C05452=1120.411,381.340,-87.972,-176.855,11.261,149.470
C05453=1120.415,381.092,-87.935,-176.859,11.258,149.470
C05454=1120.418,380.845,-87.897,-176.861,11.255,149.470
C05455=1120.423,380.598,-87.860,-176.865,11.253,149.470
C05456=1120.426,380.351,-87.822,-176.868,11.250,149.470
C05457=1120.430,380.103,-87.786,-176.871,11.248,149.471
C05458=1120.434,379.857,-87.748,-176.873,11.246,149.471
C05459=1120.437,379.609,-87.711,-176.876,11.243,149.471
C05460=1120.441,379.362,-87.673,-176.880,11.241,149.471
C05461=1120.444,379.115,-87.636,-176.883,11.238,149.471
C05462=1120.449,378.867,-87.599,-176.886,11.235,149.471
C05463=1120.452,378.621,-87.562,-176.889,11.233,149.471
C05464=1120.456,378.373,-87.524,-176.892,11.230,149.471
C05465=1120.460,378.126,-87.487,-176.895,11.228,149.472
C05466=1120.464,377.879,-87.450,-176.898,11.226,149.472
C05467=1120.467,377.631,-87.413,-176.901,11.223,149.472
C05468=1120.471,377.385,-87.375,-176.904,11.221,149.472
C05469=1120.475,377.138,-87.338,-176.908,11.218,149.472
C05470=1120.479,376.890,-87.301,-176.910,11.215,149.472
C05471=1120.482,376.643,-87.264,-176.913,11.214,149.473
C05472=1120.485,376.430,-87.232,-176.916,11.211,149.473
C05473=1120.489,376.219,-87.201,-176.919,11.209,149.473
C05474=1120.491,376.007,-87.169,-176.921,11.207,149.473
C05475=1120.495,375.795,-87.136,-176.924,11.205,149.473
C05476=1120.498,375.582,-87.105,-176.927,11.203,149.473
C05477=1120.501,375.371,-87.073,-176.929,11.201,149.473
C05478=1120.504,375.159,-87.041,-176.933,11.198,149.474
C05479=1120.508,374.946,-87.009,-176.935,11.197,149.474
C05480=1120.511,374.699,-86.973,-176.938,11.194,149.474
C05481=1120.515,374.452,-86.935,-176.941,11.191,149.474
C05482=1120.519,374.205,-86.899,-176.944,11.190,149.474
C05483=1120.523,373.957,-86.861,-176.947,11.187,149.474
C05484=1120.527,373.710,-86.824,-176.951,11.185,149.475
C05485=1120.530,373.463,-86.788,-176.954,11.182,149.475
C05486=1120.534,373.215,-86.751,-176.957,11.180,149.475
C05487=1120.538,372.968,-86.714,-176.961,11.177,149.475
C05488=1120.542,372.721,-86.677,-176.964,11.175,149.475
C05489=1120.546,372.474,-86.640,-176.967,11.173,149.476
C05490=1120.549,372.227,-86.603,-176.970,11.171,149.476
C05491=1120.552,371.980,-86.566,-176.973,11.168,149.476
C05492=1120.556,371.732,-86.529,-176.976,11.166,149.476
C05493=1120.561,371.485,-86.492,-176.980,11.163,149.477
C05494=1120.564,371.238,-86.456,-176.983,11.161,149.477
C05495=1120.567,370.990,-86.419,-176.986,11.158,149.477
C05496=1120.571,370.743,-86.382,-176.989,11.157,149.477
C05497=1120.575,370.496,-86.347,-176.992,11.154,149.477
C05498=1120.579,370.249,-86.310,-176.996,11.152,149.478
C05499=1120.583,370.001,-86.273,-176.999,11.149,149.478
C05500=1120.586,369.754,-86.236,-177.002,11.147,149.478
C05501=1120.590,369.507,-86.199,-177.005,11.144,149.478
C05502=1120.594,369.259,-86.163,-177.009,11.142,149.478
C05503=1120.598,369.012,-86.126,-177.012,11.139,149.479
C05504=1120.602,368.765,-86.089,-177.015,11.137,149.479
C05505=1120.606,368.518,-86.053,-177.018,11.135,149.479
C05506=1120.609,368.271,-86.017,-177.021,11.133,149.479
C05507=1120.613,368.023,-85.980,-177.025,11.130,149.480
C05508=1120.616,367.776,-85.944,-177.028,11.128,149.480
C05509=1120.620,367.529,-85.907,-177.032,11.125,149.480
C05510=1120.625,367.281,-85.870,-177.035,11.123,149.480
C05511=1120.628,367.034,-85.834,-177.038,11.121,149.481
C05512=1120.632,366.787,-85.797,-177.042,11.118,149.481
C05513=1120.636,366.540,-85.761,-177.045,11.116,149.481
C05514=1120.640,366.292,-85.725,-177.048,11.113,149.481
C05515=1120.643,366.044,-85.688,-177.052,11.111,149.482
C05516=1120.647,365.797,-85.651,-177.055,11.109,149.482
C05517=1120.651,365.550,-85.616,-177.058,11.107,149.482
C05518=1120.655,365.303,-85.579,-177.061,11.104,149.482
C05519=1120.658,365.056,-85.543,-177.064,11.102,149.482
C05520=1120.662,364.808,-85.507,-177.068,11.099,149.483
C05521=1120.666,364.561,-85.470,-177.071,11.097,149.483
C05522=1120.670,364.314,-85.434,-177.075,11.095,149.483
C05523=1120.674,364.066,-85.398,-177.078,11.092,149.483
C05524=1120.678,363.819,-85.361,-177.081,11.090,149.484
C05525=1120.681,363.572,-85.326,-177.085,11.087,149.484
C05526=1120.685,363.324,-85.289,-177.088,11.085,149.484
C05527=1120.689,363.077,-85.253,-177.092,11.083,149.485
C05528=1120.692,362.864,-85.222,-177.094,11.081,149.485
C05529=1120.696,362.652,-85.191,-177.098,11.079,149.485
C05530=1120.699,362.440,-85.160,-177.100,11.077,149.485
C05531=1120.702,362.228,-85.129,-177.103,11.075,149.485
C05532=1120.705,362.015,-85.098,-177.106,11.072,149.486
C05533=1120.708,361.803,-85.067,-177.109,11.071,149.486
C05534=1120.711,361.591,-85.036,-177.112,11.068,149.486
C05535=1120.715,361.379,-85.005,-177.115,11.067,149.486
C05536=1120.718,361.132,-84.969,-177.118,11.064,149.486
C05537=1120.723,360.884,-84.933,-177.121,11.062,149.487
C05538=1120.726,360.637,-84.897,-177.125,11.059,149.487
C05539=1120.730,360.390,-84.861,-177.128,11.057,149.487
C05540=1120.734,360.142,-84.825,-177.131,11.055,149.488
C05541=1120.738,359.895,-84.789,-177.135,11.052,149.488
C05542=1120.741,359.648,-84.753,-177.138,11.050,149.488
C05543=1120.745,359.400,-84.717,-177.142,11.047,149.488
C05544=1120.749,359.152,-84.681,-177.145,11.045,149.489
C05545=1120.753,358.905,-84.646,-177.148,11.043,149.489
C05546=1120.756,358.658,-84.609,-177.152,11.040,149.489
C05547=1120.761,358.410,-84.573,-177.155,11.038,149.489
C05548=1120.764,358.163,-84.538,-177.159,11.035,149.490
C05549=1120.768,357.915,-84.502,-177.162,11.033,149.490
C05550=1120.771,357.668,-84.466,-177.165,11.031,149.490
C05551=1120.775,357.421,-84.430,-177.169,11.028,149.490
C05552=1120.780,357.174,-84.395,-177.173,11.025,149.491
C05553=1120.784,356.926,-84.359,-177.176,11.023,149.491
C05554=1120.787,356.679,-84.323,-177.180,11.020,149.491
C05555=1120.791,356.431,-84.288,-177.183,11.018,149.491
C05556=1120.795,356.184,-84.252,-177.187,11.016,149.492
C05557=1120.799,355.936,-84.216,-177.190,11.013,149.492
C05558=1120.803,355.688,-84.181,-177.193,11.011,149.492
C05559=1120.806,355.441,-84.144,-177.197,11.008,149.492
C05560=1120.810,355.195,-84.109,-177.200,11.006,149.493
C05561=1120.814,354.947,-84.074,-177.204,11.004,149.493
C05562=1120.818,354.700,-84.038,-177.207,11.001,149.493
C05563=1120.821,354.452,-84.003,-177.211,10.998,149.493
C05564=1120.825,354.205,-83.967,-177.214,10.995,149.494
C05565=1120.829,353.957,-83.931,-177.217,10.993,149.494
C05566=1120.834,353.709,-83.896,-177.221,10.991,149.494
C05567=1120.838,353.462,-83.861,-177.224,10.988,149.495
C05568=1120.841,353.214,-83.825,-177.228,10.986,149.495
C05569=1120.845,352.967,-83.790,-177.231,10.983,149.495
C05570=1120.849,352.719,-83.754,-177.235,10.980,149.495
C05571=1120.852,352.472,-83.719,-177.239,10.978,149.496
C05572=1120.857,352.225,-83.683,-177.242,10.976,149.496
C05573=1120.860,351.978,-83.648,-177.245,10.973,149.496
C05574=1120.864,351.729,-83.613,-177.249,10.971,149.496
C05575=1120.868,351.482,-83.578,-177.252,10.968,149.496
C05576=1120.872,351.235,-83.542,-177.256,10.965,149.497
C05577=1120.876,350.988,-83.507,-177.259,10.963,149.497
C05578=1120.879,350.740,-83.471,-177.263,10.960,149.497
C05579=1120.883,350.492,-83.436,-177.266,10.958,149.498
C05580=1120.888,350.245,-83.401,-177.270,10.955,149.498
C05581=1120.891,349.998,-83.366,-177.273,10.952,149.498
C05582=1120.895,349.750,-83.331,-177.277,10.950,149.498
C05583=1120.899,349.502,-83.295,-177.280,10.947,149.498
C05584=1120.902,349.290,-83.266,-177.283,10.945,149.499
C05585=1120.906,349.078,-83.235,-177.286,10.943,149.499
C05586=1120.909,348.866,-83.205,-177.288,10.941,149.499
C05587=1120.912,348.652,-83.175,-177.291,10.938,149.499
C05588=1120.916,348.440,-83.145,-177.294,10.937,149.499
C05589=1120.919,348.228,-83.114,-177.297,10.935,149.500
C05590=1120.923,348.016,-83.085,-177.300,10.932,149.500
C05591=1120.926,347.803,-83.054,-177.302,10.931,149.500
C05592=1120.929,347.556,-83.019,-177.306,10.928,149.500
C05593=1120.933,347.308,-82.985,-177.309,10.926,149.500
C05594=1120.938,347.061,-82.949,-177.312,10.923,149.500
C05595=1120.942,346.813,-82.915,-177.315,10.920,149.501
C05596=1120.945,346.566,-82.879,-177.318,10.918,149.501
C05597=1120.950,346.318,-82.845,-177.322,10.915,149.501
C05598=1120.953,346.071,-82.810,-177.325,10.913,149.501
C05599=1120.957,345.823,-82.775,-177.328,10.911,149.501
C05600=1120.961,345.576,-82.740,-177.331,10.908,149.502
C05601=1120.965,345.328,-82.705,-177.335,10.905,149.502
C05602=1120.969,345.080,-82.670,-177.337,10.904,149.502
C05603=1120.972,344.833,-82.635,-177.341,10.901,149.502
C05604=1120.976,344.585,-82.601,-177.344,10.899,149.502
C05605=1120.981,344.338,-82.565,-177.347,10.896,149.503
C05606=1120.985,344.090,-82.531,-177.350,10.893,149.503
C05607=1120.988,343.843,-82.497,-177.353,10.891,149.503
C05608=1120.992,343.596,-82.461,-177.357,10.889,149.503
C05609=1120.996,343.348,-82.426,-177.360,10.886,149.503
C05610=1121.001,343.100,-82.392,-177.363,10.884,149.504
C05611=1121.004,342.852,-82.358,-177.367,10.881,149.504
C05612=1121.008,342.606,-82.322,-177.370,10.878,149.504
C05613=1121.012,342.357,-82.288,-177.373,10.876,149.504
C05614=1121.016,342.110,-82.254,-177.376,10.873,149.504
C05615=1121.020,341.862,-82.219,-177.380,10.871,149.505
C05616=1121.024,341.615,-82.183,-177.383,10.869,149.505
C05617=1121.027,341.368,-82.149,-177.385,10.867,149.505
C05618=1121.031,341.120,-82.115,-177.388,10.864,149.505
C05619=1121.036,340.872,-82.080,-177.392,10.862,149.505
C05620=1121.039,340.624,-82.046,-177.395,10.859,149.506
C05621=1121.043,340.377,-82.011,-177.398,10.857,149.506
C05622=1121.047,340.129,-81.976,-177.401,10.854,149.506
C05623=1121.051,339.882,-81.942,-177.405,10.851,149.506
C05624=1121.055,339.634,-81.907,-177.408,10.849,149.506
C05625=1121.059,339.387,-81.873,-177.411,10.847,149.507
C05626=1121.063,339.139,-81.838,-177.414,10.844,149.507
C05627=1121.068,338.891,-81.804,-177.417,10.841,149.507
C05628=1121.071,338.644,-81.770,-177.421,10.839,149.507
C05629=1121.075,338.396,-81.735,-177.424,10.836,149.507
C05630=1121.079,338.149,-81.701,-177.427,10.834,149.508
C05631=1121.083,337.901,-81.667,-177.430,10.831,149.508
C05632=1121.087,337.654,-81.633,-177.433,10.830,149.508
C05633=1121.091,337.406,-81.598,-177.436,10.827,149.508
C05634=1121.095,337.159,-81.564,-177.440,10.825,149.508
C05635=1121.099,336.911,-81.529,-177.443,10.822,149.508
C05636=1121.103,336.663,-81.495,-177.446,10.819,149.509
C05637=1121.107,336.415,-81.460,-177.449,10.817,149.509
C05638=1121.110,336.168,-81.427,-177.453,10.814,149.509
C05639=1121.115,335.921,-81.392,-177.455,10.812,149.509
C05640=1121.119,335.708,-81.363,-177.458,10.810,149.510
C05641=1121.122,335.496,-81.334,-177.461,10.807,149.510
C05642=1121.125,335.283,-81.305,-177.464,10.806,149.510
C05643=1121.128,335.070,-81.275,-177.467,10.803,149.510
C05644=1121.131,334.858,-81.245,-177.469,10.801,149.510
C05645=1121.135,334.645,-81.216,-177.472,10.799,149.510
C05646=1121.138,334.432,-81.187,-177.475,10.797,149.510
C05647=1121.141,334.220,-81.158,-177.477,10.795,149.511
C05648=1121.145,333.972,-81.124,-177.481,10.792,149.511
C05649=1121.150,333.725,-81.089,-177.484,10.790,149.511
C05650=1121.153,333.477,-81.056,-177.487,10.787,149.511
C05651=1121.158,333.229,-81.022,-177.490,10.784,149.511
C05652=1121.162,332.982,-80.988,-177.493,10.782,149.512
C05653=1121.165,332.734,-80.953,-177.497,10.780,149.512
C05654=1121.170,332.486,-80.920,-177.500,10.777,149.512
C05655=1121.174,332.239,-80.886,-177.502,10.775,149.512
C05656=1121.177,331.991,-80.852,-177.506,10.773,149.512
C05657=1121.181,331.744,-80.818,-177.509,10.770,149.513
C05658=1121.186,331.496,-80.784,-177.512,10.767,149.513
C05659=1121.189,331.248,-80.750,-177.515,10.765,149.513
C05660=1121.193,331.001,-80.717,-177.519,10.763,149.513
C05661=1121.198,330.753,-80.682,-177.522,10.760,149.513
C05662=1121.201,330.505,-80.649,-177.525,10.757,149.513
C05663=1121.205,330.258,-80.615,-177.528,10.755,149.514
C05664=1121.209,330.010,-80.582,-177.531,10.752,149.514
C05665=1121.213,329.762,-80.547,-177.534,10.750,149.514
C05666=1121.217,329.514,-80.514,-177.538,10.747,149.514
C05667=1121.221,329.267,-80.480,-177.541,10.745,149.515
C05668=1121.225,329.019,-80.446,-177.544,10.742,149.515
C05669=1121.228,328.771,-80.412,-177.547,10.740,149.515
C05670=1121.233,328.523,-80.379,-177.550,10.738,149.515
C05671=1121.237,328.276,-80.345,-177.553,10.735,149.515
C05672=1121.241,328.029,-80.311,-177.556,10.733,149.515
C05673=1121.244,327.781,-80.277,-177.560,10.730,149.516
C05674=1121.249,327.533,-80.244,-177.563,10.728,149.516
C05675=1121.253,327.285,-80.211,-177.566,10.725,149.516
C05676=1121.257,327.038,-80.176,-177.569,10.723,149.516
C05677=1121.261,326.789,-80.143,-177.572,10.720,149.516
C05678=1121.265,326.542,-80.110,-177.575,10.717,149.516
C05679=1121.269,326.295,-80.076,-177.579,10.715,149.517
C05680=1121.273,326.047,-80.043,-177.582,10.712,149.517
C05681=1121.277,325.799,-80.010,-177.585,10.710,149.517
C05682=1121.280,325.551,-79.975,-177.588,10.707,149.517
C05683=1121.284,325.304,-79.942,-177.592,10.705,149.518
C05684=1121.289,325.056,-79.909,-177.594,10.703,149.518
C05685=1121.293,324.808,-79.876,-177.597,10.700,149.518
C05686=1121.297,324.561,-79.842,-177.601,10.698,149.518
C05687=1121.300,324.313,-79.809,-177.604,10.695,149.518
C05688=1121.305,324.065,-79.775,-177.607,10.693,149.518
C05689=1121.309,323.817,-79.742,-177.610,10.690,149.519
C05690=1121.313,323.569,-79.708,-177.613,10.688,149.519
C05691=1121.317,323.322,-79.675,-177.616,10.685,149.519
C05692=1121.321,323.074,-79.641,-177.620,10.682,149.519
C05693=1121.324,322.826,-79.608,-177.623,10.680,149.519
C05694=1121.328,322.578,-79.575,-177.626,10.677,149.520
C05695=1121.332,322.331,-79.542,-177.629,10.675,149.520
C05696=1121.336,322.118,-79.513,-177.632,10.673,149.520
C05697=1121.340,321.906,-79.485,-177.634,10.671,149.520
C05698=1121.343,321.693,-79.456,-177.637,10.668,149.520
C05699=1121.346,321.480,-79.428,-177.639,10.666,149.520
C05700=1121.350,321.267,-79.399,-177.643,10.664,149.521
C05701=1121.353,321.054,-79.371,-177.645,10.662,149.521
C05702=1121.357,320.842,-79.343,-177.648,10.660,149.521
C05703=1121.360,320.629,-79.314,-177.651,10.658,149.521
C05704=1121.364,320.382,-79.281,-177.654,10.655,149.521
C05705=1121.368,320.134,-79.248,-177.656,10.653,149.521
C05706=1121.372,319.886,-79.215,-177.660,10.651,149.522
C05707=1121.376,319.638,-79.181,-177.663,10.648,149.522
C05708=1121.380,319.390,-79.148,-177.666,10.645,149.522
C05709=1121.384,319.142,-79.115,-177.669,10.643,149.522
C05710=1121.387,318.895,-79.082,-177.672,10.640,149.522
C05711=1121.391,318.647,-79.049,-177.675,10.638,149.523
C05712=1121.396,318.399,-79.017,-177.679,10.635,149.523
C05713=1121.400,318.151,-78.984,-177.682,10.633,149.523
C05714=1121.404,317.903,-78.951,-177.685,10.630,149.523
C05715=1121.408,317.656,-78.917,-177.688,10.628,149.523
C05716=1121.412,317.408,-78.885,-177.691,10.625,149.523
C05717=1121.416,317.160,-78.852,-177.695,10.622,149.524
C05718=1121.420,316.912,-78.819,-177.698,10.620,149.524
C05719=1121.424,316.664,-78.786,-177.700,10.618,149.524
C05720=1121.428,316.417,-78.754,-177.704,10.616,149.524
C05721=1121.432,316.169,-78.720,-177.706,10.613,149.524
C05722=1121.436,315.922,-78.687,-177.710,10.610,149.525
C05723=1121.441,315.673,-78.655,-177.713,10.608,149.525
C05724=1121.444,315.426,-78.622,-177.716,10.605,149.525
C05725=1121.448,315.178,-78.589,-177.719,10.603,149.525
C05726=1121.453,314.930,-78.557,-177.722,10.600,149.525
C05727=1121.456,314.682,-78.524,-177.726,10.597,149.526
C05728=1121.460,314.435,-78.491,-177.729,10.595,149.526
C05729=1121.465,314.186,-78.458,-177.732,10.592,149.526
C05730=1121.468,313.939,-78.426,-177.735,10.590,149.526
C05731=1121.472,313.691,-78.393,-177.738,10.587,149.526
C05732=1121.477,313.443,-78.360,-177.741,10.585,149.526
C05733=1121.480,313.195,-78.328,-177.744,10.583,149.527
C05734=1121.484,312.947,-78.295,-177.747,10.580,149.527
C05735=1121.489,312.700,-78.263,-177.750,10.578,149.527
C05736=1121.493,312.452,-78.231,-177.753,10.575,149.527
C05737=1121.497,312.204,-78.198,-177.757,10.573,149.527
C05738=1121.501,311.956,-78.166,-177.760,10.570,149.527
C05739=1121.505,311.708,-78.133,-177.763,10.567,149.528
C05740=1121.509,311.460,-78.100,-177.766,10.565,149.528
C05741=1121.513,311.213,-78.068,-177.769,10.562,149.528
C05742=1121.517,310.964,-78.035,-177.773,10.560,149.528
C05743=1121.520,310.717,-78.003,-177.775,10.557,149.528
C05744=1121.525,310.468,-77.970,-177.778,10.555,149.529
C05745=1121.529,310.222,-77.938,-177.781,10.552,149.529
C05746=1121.533,309.973,-77.905,-177.784,10.550,149.529
C05747=1121.537,309.725,-77.874,-177.787,10.547,149.529
C05748=1121.541,309.478,-77.840,-177.791,10.545,149.529
C05749=1121.545,309.230,-77.809,-177.794,10.542,149.530
C05750=1121.549,308.981,-77.776,-177.797,10.540,149.530
C05751=1121.553,308.735,-77.744,-177.800,10.537,149.530
C05752=1121.557,308.521,-77.716,-177.803,10.535,149.530
C05753=1121.560,308.308,-77.688,-177.805,10.532,149.530
C05754=1121.564,308.095,-77.661,-177.808,10.531,149.530
C05755=1121.568,307.882,-77.633,-177.810,10.529,149.530
C05756=1121.571,307.670,-77.605,-177.813,10.526,149.531
C05757=1121.574,307.457,-77.577,-177.816,10.524,149.531
C05758=1121.578,307.244,-77.550,-177.818,10.522,149.531
C05759=1121.582,307.031,-77.522,-177.821,10.520,149.531
C05760=1121.585,306.783,-77.490,-177.825,10.517,149.531
C05761=1121.590,306.535,-77.459,-177.828,10.514,149.531
C05762=1121.594,306.288,-77.425,-177.831,10.512,149.532
C05763=1121.598,306.040,-77.394,-177.834,10.510,149.532
C05764=1121.602,305.791,-77.361,-177.837,10.508,149.532
C05765=1121.606,305.543,-77.329,-177.840,10.505,149.532
C05766=1121.610,305.296,-77.298,-177.843,10.502,149.532
C05767=1121.615,305.048,-77.265,-177.846,10.500,149.533
C05768=1121.618,304.800,-77.234,-177.849,10.497,149.533
C05769=1121.622,304.553,-77.201,-177.852,10.495,149.533
C05770=1121.627,304.304,-77.169,-177.855,10.492,149.533
C05771=1121.630,304.056,-77.137,-177.859,10.489,149.533
C05772=1121.634,303.808,-77.105,-177.862,10.487,149.533
C05773=1121.639,303.561,-77.073,-177.865,10.484,149.534
C05774=1121.643,303.313,-77.041,-177.868,10.482,149.534
C05775=1121.647,303.065,-77.010,-177.871,10.480,149.534
C05776=1121.652,302.817,-76.977,-177.873,10.477,149.534
C05777=1121.655,302.569,-76.946,-177.877,10.475,149.534
C05778=1121.659,302.321,-76.914,-177.880,10.472,149.535
C05779=1121.664,302.073,-76.882,-177.883,10.469,149.535
C05780=1121.668,301.825,-76.850,-177.886,10.467,149.535
C05781=1121.672,301.577,-76.819,-177.889,10.464,149.535
C05782=1121.676,301.329,-76.787,-177.893,10.462,149.535
C05783=1121.681,301.081,-76.755,-177.896,10.459,149.535
C05784=1121.684,300.833,-76.723,-177.899,10.457,149.536
C05785=1121.689,300.586,-76.691,-177.902,10.454,149.536
C05786=1121.692,300.337,-76.660,-177.905,10.451,149.536
C05787=1121.696,300.089,-76.628,-177.908,10.449,149.536
C05788=1121.701,299.842,-76.596,-177.911,10.447,149.536
C05789=1121.705,299.593,-76.565,-177.914,10.444,149.536
C05790=1121.709,299.345,-76.533,-177.917,10.442,149.537
C05791=1121.713,299.098,-76.501,-177.920,10.439,149.537
C05792=1121.717,298.850,-76.469,-177.923,10.437,149.537
C05793=1121.721,298.602,-76.439,-177.926,10.434,149.537
C05794=1121.725,298.354,-76.407,-177.930,10.431,149.537
C05795=1121.729,298.106,-76.375,-177.933,10.429,149.537
C05796=1121.734,297.858,-76.343,-177.936,10.426,149.538
C05797=1121.738,297.609,-76.312,-177.939,10.423,149.538
C05798=1121.742,297.362,-76.280,-177.942,10.422,149.538
C05799=1121.746,297.114,-76.248,-177.945,10.419,149.538
C05800=1121.750,296.865,-76.217,-177.948,10.417,149.538
C05801=1121.754,296.618,-76.186,-177.951,10.414,149.539
C05802=1121.758,296.370,-76.154,-177.954,10.411,149.539
C05803=1121.762,296.122,-76.123,-177.957,10.409,149.539
C05804=1121.766,295.874,-76.091,-177.960,10.406,149.539
C05805=1121.771,295.626,-76.061,-177.963,10.403,149.539
C05806=1121.774,295.378,-76.029,-177.967,10.401,149.540
C05807=1121.779,295.130,-75.998,-177.970,10.398,149.540
C05808=1121.783,294.904,-75.969,-177.972,10.396,149.540
C05809=1121.786,294.679,-75.940,-177.975,10.394,149.540
C05810=1121.790,294.454,-75.912,-177.978,10.392,149.540
C05811=1121.794,294.228,-75.883,-177.980,10.389,149.540
C05812=1121.797,294.003,-75.855,-177.983,10.387,149.541
C05813=1121.801,293.778,-75.827,-177.986,10.385,149.541
C05814=1121.805,293.552,-75.798,-177.988,10.383,149.541
C05815=1121.809,293.327,-75.770,-177.992,10.380,149.541
C05816=1121.813,293.079,-75.739,-177.995,10.378,149.541
C05817=1121.817,292.831,-75.708,-177.998,10.375,149.541
C05818=1121.821,292.583,-75.676,-178.001,10.372,149.541
C05819=1121.825,292.335,-75.646,-178.004,10.370,149.542
C05820=1121.829,292.099,-75.616,-178.007,10.368,149.542
C05821=1121.833,291.863,-75.586,-178.010,10.365,149.542
C05822=1121.837,291.628,-75.556,-178.013,10.363,149.542
C05823=1121.841,291.393,-75.527,-178.015,10.361,149.542
C05824=1121.845,291.157,-75.497,-178.018,10.358,149.543
C05825=1121.848,290.921,-75.467,-178.021,10.356,149.543
C05826=1121.853,290.685,-75.438,-178.024,10.353,149.543
C05827=1121.856,290.450,-75.409,-178.027,10.351,149.543
C05828=1121.861,290.202,-75.378,-178.030,10.348,149.543
C05829=1121.865,289.953,-75.347,-178.033,10.346,149.543
C05830=1121.869,289.706,-75.316,-178.036,10.343,149.543
C05831=1121.873,289.457,-75.284,-178.040,10.341,149.544
C05832=1121.877,289.210,-75.254,-178.043,10.338,149.544
C05833=1121.881,288.962,-75.223,-178.045,10.335,149.544
C05834=1121.886,288.713,-75.192,-178.049,10.333,149.544
C05835=1121.890,288.466,-75.161,-178.051,10.331,149.544
C05836=1121.894,288.217,-75.130,-178.054,10.328,149.545
C05837=1121.898,287.969,-75.100,-178.057,10.326,149.545
C05838=1121.902,287.721,-75.069,-178.061,10.323,149.545
C05839=1121.906,287.473,-75.038,-178.064,10.320,149.545
C05840=1121.910,287.225,-75.008,-178.067,10.318,149.545
C05841=1121.914,286.976,-74.976,-178.070,10.315,149.545
C05842=1121.919,286.729,-74.945,-178.073,10.313,149.546
C05843=1121.923,286.481,-74.914,-178.076,10.310,149.546
C05844=1121.926,286.233,-74.884,-178.079,10.307,149.546
C05845=1121.931,285.985,-74.853,-178.082,10.306,149.546
C05846=1121.936,285.737,-74.822,-178.085,10.303,149.546
C05847=1121.939,285.489,-74.792,-178.088,10.301,149.547
C05848=1121.944,285.241,-74.761,-178.091,10.298,149.547
C05849=1121.948,284.993,-74.730,-178.094,10.295,149.547
C05850=1121.951,284.744,-74.699,-178.097,10.293,149.547
C05851=1121.956,284.496,-74.669,-178.100,10.290,149.547
C05852=1121.960,284.249,-74.639,-178.104,10.287,149.547
C05853=1121.965,284.001,-74.608,-178.107,10.285,149.547
C05854=1121.969,283.752,-74.577,-178.109,10.283,149.548
C05855=1121.973,283.504,-74.547,-178.112,10.280,149.548
C05856=1121.977,283.256,-74.516,-178.115,10.277,149.548
C05857=1121.981,283.007,-74.486,-178.119,10.275,149.548
C05858=1121.985,282.759,-74.455,-178.121,10.272,149.548
C05859=1121.990,282.512,-74.424,-178.125,10.270,149.549
C05860=1121.994,282.264,-74.394,-178.128,10.267,149.549
C05861=1121.998,282.015,-74.363,-178.131,10.264,149.549
C05862=1122.002,281.767,-74.334,-178.134,10.262,149.549
C05863=1122.007,281.519,-74.303,-178.136,10.260,149.549
C05864=1122.010,281.306,-74.277,-178.140,10.258,149.550
C05865=1122.014,281.093,-74.250,-178.143,10.255,149.550
C05866=1122.017,280.880,-74.225,-178.145,10.253,149.550
C05867=1122.021,280.666,-74.198,-178.148,10.250,149.550
C05868=1122.024,280.453,-74.173,-178.151,10.248,149.550
C05869=1122.028,280.240,-74.146,-178.154,10.246,149.550
C05870=1122.031,280.027,-74.120,-178.157,10.243,149.551
C05871=1122.036,279.813,-74.094,-178.160,10.240,149.551
C05872=1122.039,279.566,-74.064,-178.163,10.238,149.551
C05873=1122.043,279.318,-74.034,-178.166,10.235,149.551
C05874=1122.048,279.070,-74.004,-178.169,10.233,149.551
C05875=1122.051,278.821,-73.973,-178.172,10.230,149.551
C05876=1122.056,278.573,-73.943,-178.176,10.227,149.552
C05877=1122.060,278.325,-73.913,-178.179,10.224,149.552
C05878=1122.064,278.077,-73.883,-178.183,10.222,149.552
C05879=1122.069,277.829,-73.853,-178.186,10.219,149.552
C05880=1122.072,277.580,-73.822,-178.188,10.216,149.552
C05881=1122.077,277.332,-73.792,-178.192,10.214,149.553
C05882=1122.081,277.084,-73.762,-178.195,10.211,149.553
C05883=1122.085,276.837,-73.732,-178.198,10.208,149.553
C05884=1122.090,276.588,-73.702,-178.201,10.206,149.553
C05885=1122.094,276.340,-73.672,-178.205,10.202,149.553
C05886=1122.098,276.092,-73.642,-178.208,10.200,149.553
C05887=1122.102,275.844,-73.612,-178.211,10.197,149.553
C05888=1122.106,275.595,-73.582,-178.214,10.194,149.554
C05889=1122.110,275.347,-73.552,-178.217,10.192,149.554
C05890=1122.114,275.099,-73.522,-178.220,10.189,149.554
C05891=1122.119,274.851,-73.492,-178.223,10.186,149.554
C05892=1122.123,274.603,-73.462,-178.226,10.184,149.554
C05893=1122.127,274.355,-73.433,-178.229,10.181,149.554
C05894=1122.131,274.106,-73.403,-178.232,10.178,149.554
C05895=1122.136,273.858,-73.372,-178.235,10.175,149.554
C05896=1122.140,273.610,-73.343,-178.238,10.173,149.555
C05897=1122.144,273.362,-73.313,-178.241,10.170,149.555
C05898=1122.148,273.114,-73.283,-178.243,10.168,149.555
C05899=1122.152,272.866,-73.254,-178.246,10.165,149.555
C05900=1122.157,272.617,-73.224,-178.249,10.163,149.555
C05901=1122.161,272.369,-73.193,-178.252,10.160,149.555
C05902=1122.165,272.121,-73.164,-178.255,10.157,149.555
C05903=1122.169,271.873,-73.134,-178.258,10.154,149.555
C05904=1122.173,271.624,-73.105,-178.261,10.152,149.556
C05905=1122.177,271.376,-73.075,-178.264,10.149,149.556
C05906=1122.182,271.128,-73.045,-178.266,10.147,149.556
C05907=1122.186,270.880,-73.015,-178.269,10.144,149.556
C05908=1122.190,270.632,-72.986,-178.272,10.141,149.556
C05909=1122.195,270.383,-72.956,-178.275,10.139,149.556
C05910=1122.199,270.135,-72.927,-178.278,10.136,149.556
C05911=1122.203,269.887,-72.897,-178.280,10.134,149.556
C05912=1122.207,269.639,-72.867,-178.283,10.131,149.556
C05913=1122.211,269.391,-72.838,-178.286,10.128,149.556
C05914=1122.216,269.143,-72.809,-178.289,10.126,149.557
C05915=1122.220,268.895,-72.779,-178.291,10.124,149.557
C05916=1122.224,268.647,-72.750,-178.294,10.121,149.557
C05917=1122.229,268.398,-72.720,-178.297,10.118,149.557
C05918=1122.233,268.150,-72.690,-178.300,10.116,149.557
C05919=1122.237,267.902,-72.661,-178.303,10.113,149.557
C05920=1122.241,267.688,-72.636,-178.305,10.111,149.557
C05921=1122.244,267.475,-72.610,-178.307,10.109,149.557
C05922=1122.248,267.261,-72.585,-178.309,10.107,149.558
C05923=1122.251,267.049,-72.559,-178.311,10.105,149.557
C05924=1122.255,266.835,-72.534,-178.314,10.103,149.558
C05925=1122.258,266.622,-72.509,-178.316,10.101,149.558
C05926=1122.263,266.409,-72.484,-178.319,10.098,149.558
C05927=1122.266,266.196,-72.459,-178.321,10.096,149.558
C05928=1122.270,265.947,-72.430,-178.323,10.094,149.558
C05929=1122.275,265.699,-72.400,-178.326,10.091,149.558
C05930=1122.279,265.451,-72.371,-178.328,10.089,149.558
C05931=1122.283,265.203,-72.341,-178.331,10.087,149.558
C05932=1122.287,264.954,-72.312,-178.334,10.085,149.558
C05933=1122.292,264.705,-72.283,-178.337,10.082,149.558
C05934=1122.296,264.457,-72.254,-178.339,10.080,149.559
C05935=1122.301,264.210,-72.224,-178.343,10.077,149.559
C05936=1122.305,263.961,-72.195,-178.346,10.074,149.559
C05937=1122.309,263.713,-72.166,-178.350,10.071,149.559
C05938=1122.313,263.464,-72.137,-178.353,10.068,149.560
C05939=1122.317,263.216,-72.108,-178.357,10.065,149.560
C05940=1122.321,262.968,-72.078,-178.360,10.062,149.560
C05941=1122.326,262.720,-72.049,-178.364,10.059,149.560
C05942=1122.330,262.471,-72.021,-178.367,10.056,149.560
C05943=1122.334,262.223,-71.991,-178.371,10.053,149.560
C05944=1122.339,261.975,-71.962,-178.374,10.050,149.560
C05945=1122.342,261.726,-71.934,-178.377,10.047,149.561
C05946=1122.347,261.479,-71.905,-178.380,10.044,149.561
C05947=1122.351,261.231,-71.875,-178.383,10.042,149.561
C05948=1122.356,260.982,-71.846,-178.387,10.038,149.561
C05949=1122.360,260.733,-71.817,-178.390,10.036,149.561
C05950=1122.363,260.485,-71.788,-178.393,10.033,149.561
C05951=1122.369,260.237,-71.760,-178.397,10.029,149.562
C05952=1122.373,259.989,-71.730,-178.400,10.027,149.562
C05953=1122.377,259.740,-71.701,-178.403,10.024,149.562
C05954=1122.381,259.492,-71.673,-178.406,10.021,149.562
C05955=1122.386,259.244,-71.644,-178.409,10.017,149.562
C05956=1122.390,258.996,-71.615,-178.412,10.015,149.562
C05957=1122.394,258.747,-71.587,-178.415,10.012,149.562
C05958=1122.398,258.499,-71.557,-178.418,10.009,149.562
C05959=1122.403,258.251,-71.529,-178.421,10.006,149.562
C05960=1122.406,258.003,-71.500,-178.424,10.004,149.563
C05961=1122.411,257.754,-71.471,-178.427,10.001,149.563
C05962=1122.415,257.505,-71.442,-178.430,9.998,149.563
C05963=1122.419,257.258,-71.414,-178.433,9.995,149.563
C05964=1122.424,257.009,-71.385,-178.435,9.992,149.563
C05965=1122.428,256.760,-71.356,-178.439,9.989,149.563
C05966=1122.432,256.513,-71.328,-178.441,9.987,149.563
C05967=1122.437,256.264,-71.299,-178.444,9.984,149.563
C05968=1122.441,256.015,-71.270,-178.447,9.981,149.563
C05969=1122.445,255.768,-71.242,-178.448,9.979,149.563
C05970=1122.450,255.519,-71.213,-178.448,9.978,149.563
C05971=1122.453,255.271,-71.184,-178.448,9.977,149.563
C05972=1122.458,255.023,-71.156,-178.449,9.975,149.562
C05973=1122.462,254.775,-71.127,-178.450,9.974,149.562
C05974=1122.466,254.526,-71.098,-178.452,9.972,149.562
C05975=1122.471,254.277,-71.070,-178.453,9.971,149.562
C05976=1122.474,254.064,-71.046,-178.454,9.969,149.562
C05977=1122.478,253.850,-71.021,-178.455,9.967,149.562
C05978=1122.482,253.638,-70.996,-178.457,9.966,149.562
C05979=1122.485,253.424,-70.972,-178.458,9.965,149.562
C05980=1122.489,253.210,-70.947,-178.460,9.962,149.562
C05981=1122.494,252.997,-70.923,-178.462,9.961,149.562
C05982=1122.497,252.784,-70.898,-178.464,9.959,149.562
C05983=1122.500,252.570,-70.874,-178.467,9.957,149.563
C05984=1122.505,252.322,-70.845,-178.470,9.954,149.563
C05985=1122.509,252.074,-70.817,-178.472,9.952,149.563
C05986=1122.513,251.825,-70.788,-178.475,9.950,149.563
C05987=1122.518,251.577,-70.760,-178.478,9.947,149.563
C05988=1122.522,251.328,-70.732,-178.482,9.944,149.564
C05989=1122.526,251.081,-70.703,-178.485,9.941,149.564
C05990=1122.531,250.832,-70.674,-178.489,9.938,149.564
C05991=1122.534,250.583,-70.646,-178.493,9.935,149.564
C05992=1122.539,250.335,-70.618,-178.497,9.932,149.564
C05993=1122.543,250.087,-70.590,-178.501,9.929,149.565
C05994=1122.548,249.839,-70.562,-178.506,9.925,149.565
C05995=1122.552,249.590,-70.533,-178.510,9.922,149.566
C05996=1122.556,249.342,-70.505,-178.515,9.918,149.566
C05997=1122.561,249.093,-70.477,-178.519,9.914,149.566
C05998=1122.565,248.845,-70.448,-178.525,9.910,149.567
C05999=1122.569,248.597,-70.421,-178.530,9.906,149.567
C06000=1122.573,248.348,-70.392,-178.535,9.901,149.567
C06001=1122.578,248.100,-70.364,-178.541,9.897,149.568
C06002=1122.582,247.851,-70.336,-178.546,9.892,149.568
C06003=1122.587,247.603,-70.308,-178.553,9.887,149.568
C06004=1122.590,247.355,-70.280,-178.557,9.884,149.569
C06005=1122.595,247.106,-70.252,-178.558,9.881,149.568
C06006=1122.599,246.858,-70.225,-178.560,9.879,149.568
C06007=1122.604,246.609,-70.196,-178.561,9.877,149.568
C06008=1122.608,246.362,-70.168,-178.563,9.875,149.568
C06009=1122.612,246.113,-70.140,-178.565,9.872,149.568
C06010=1122.616,245.865,-70.112,-178.566,9.870,149.568
C06011=1122.621,245.616,-70.084,-178.568,9.867,149.568
C06012=1122.625,245.368,-70.056,-178.570,9.865,149.568
C06013=1122.629,245.119,-70.028,-178.572,9.863,149.568
C06014=1122.634,244.871,-70.001,-178.574,9.860,149.568
C06015=1122.638,244.623,-69.973,-178.576,9.858,149.567
C06016=1122.643,244.374,-69.945,-178.577,9.856,149.567
C06017=1122.647,244.126,-69.917,-178.579,9.853,149.567
C06018=1122.651,243.877,-69.890,-178.581,9.851,149.567
C06019=1122.655,243.629,-69.862,-178.583,9.849,149.567
C06020=1122.659,243.380,-69.834,-178.585,9.846,149.567
C06021=1122.664,243.132,-69.805,-178.587,9.844,149.567
C06022=1122.669,242.884,-69.778,-178.589,9.842,149.567
C06023=1122.673,242.635,-69.750,-178.592,9.839,149.567
C06024=1122.677,242.387,-69.723,-178.594,9.837,149.567
C06025=1122.681,242.138,-69.695,-178.596,9.835,149.567
C06026=1122.685,241.890,-69.667,-178.598,9.832,149.567
C06027=1122.690,241.642,-69.640,-178.600,9.830,149.567
C06028=1122.695,241.393,-69.611,-178.603,9.827,149.567
C06029=1122.699,241.145,-69.583,-178.605,9.825,149.567
C06030=1122.704,240.896,-69.556,-178.607,9.823,149.567
C06031=1122.707,240.648,-69.528,-178.609,9.820,149.567
C06032=1122.711,240.435,-69.505,-178.612,9.818,149.567
C06033=1122.715,240.220,-69.482,-178.614,9.815,149.567
C06034=1122.719,240.007,-69.458,-178.616,9.813,149.568
C06035=1122.722,239.793,-69.434,-178.617,9.812,149.567
C06036=1122.726,239.580,-69.410,-178.620,9.810,149.568
C06037=1122.730,239.366,-69.386,-178.621,9.808,149.568
C06038=1122.734,239.153,-69.362,-178.624,9.806,149.568
C06039=1122.738,238.940,-69.339,-178.626,9.803,149.568
C06040=1122.741,238.691,-69.311,-178.629,9.801,149.568
C06041=1122.746,238.443,-69.284,-178.632,9.798,149.568
C06042=1122.750,238.195,-69.256,-178.633,9.795,149.568
C06043=1122.754,237.945,-69.229,-178.636,9.793,149.568
C06044=1122.759,237.698,-69.201,-178.639,9.790,149.568
C06045=1122.763,237.449,-69.174,-178.642,9.788,149.568
C06046=1122.767,237.200,-69.147,-178.644,9.785,149.568
C06047=1122.772,236.952,-69.119,-178.647,9.782,149.568
C06048=1122.776,236.704,-69.092,-178.650,9.779,149.568
C06049=1122.781,236.456,-69.064,-178.652,9.777,149.569
C06050=1122.785,236.206,-69.037,-178.655,9.775,149.569
C06051=1122.790,235.958,-69.010,-178.658,9.772,149.569
C06052=1122.794,235.710,-68.982,-178.661,9.769,149.569
C06053=1122.798,235.461,-68.954,-178.664,9.766,149.569
C06054=1122.803,235.212,-68.927,-178.667,9.763,149.569
C06055=1122.807,234.964,-68.900,-178.670,9.761,149.569
C06056=1122.812,234.716,-68.873,-178.673,9.758,149.569
C06057=1122.816,234.467,-68.845,-178.675,9.755,149.569
C06058=1122.820,234.219,-68.819,-178.678,9.752,149.569
C06059=1122.824,233.970,-68.792,-178.681,9.750,149.570
C06060=1122.829,233.722,-68.764,-178.684,9.747,149.570
C06061=1122.833,233.474,-68.737,-178.687,9.744,149.570
C06062=1122.837,233.225,-68.709,-178.690,9.741,149.570
C06063=1122.842,232.976,-68.682,-178.694,9.738,149.570
C06064=1122.847,232.728,-68.655,-178.697,9.735,149.570
C06065=1122.850,232.480,-68.628,-178.700,9.732,149.570
C06066=1122.855,232.232,-68.601,-178.703,9.729,149.570
C06067=1122.859,231.982,-68.573,-178.706,9.726,149.571
C06068=1122.864,231.734,-68.546,-178.709,9.723,149.571
C06069=1122.868,231.485,-68.519,-178.713,9.720,149.571
C06070=1122.872,231.237,-68.493,-178.716,9.717,149.571
C06071=1122.877,230.989,-68.466,-178.719,9.714,149.571
C06072=1122.881,230.740,-68.439,-178.722,9.711,149.571
C06073=1122.886,230.491,-68.411,-178.726,9.707,149.571
C06074=1122.889,230.243,-68.385,-178.729,9.705,149.571
C06075=1122.894,229.994,-68.358,-178.732,9.701,149.572
C06076=1122.899,229.746,-68.331,-178.736,9.697,149.572
C06077=1122.903,229.498,-68.304,-178.739,9.694,149.572
C06078=1122.907,229.249,-68.277,-178.742,9.691,149.572
C06079=1122.912,229.001,-68.250,-178.746,9.688,149.572
C06080=1122.916,228.752,-68.224,-178.750,9.684,149.572
C06081=1122.921,228.504,-68.197,-178.753,9.681,149.572
C06082=1122.925,228.255,-68.170,-178.756,9.678,149.572
C06083=1122.929,228.006,-68.143,-178.759,9.675,149.572
C06084=1122.933,227.757,-68.116,-178.762,9.671,149.572
C06085=1122.938,227.509,-68.089,-178.766,9.668,149.573
C06086=1122.942,227.261,-68.063,-178.769,9.665,149.573
C06087=1122.947,227.012,-68.036,-178.772,9.661,149.573
C06088=1122.951,226.799,-68.013,-178.774,9.659,149.573
C06089=1122.955,226.585,-67.990,-178.777,9.656,149.573
C06090=1122.958,226.372,-67.968,-178.780,9.653,149.573
C06091=1122.962,226.157,-67.945,-178.782,9.650,149.573
C06092=1122.966,225.944,-67.922,-178.785,9.647,149.573
C06093=1122.969,225.731,-67.899,-178.788,9.644,149.573
C06094=1122.973,225.517,-67.876,-178.790,9.642,149.573
C06095=1122.977,225.303,-67.853,-178.793,9.639,149.573
C06096=1122.982,225.054,-67.827,-178.796,9.635,149.573
C06097=1122.986,224.806,-67.800,-178.798,9.632,149.573
C06098=1122.990,224.558,-67.774,-178.801,9.630,149.573
C06099=1122.995,224.309,-67.747,-178.804,9.626,149.573
C06100=1122.999,224.061,-67.721,-178.807,9.623,149.573
C06101=1123.004,223.812,-67.694,-178.810,9.620,149.573
C06102=1123.008,223.563,-67.668,-178.812,9.617,149.573
C06103=1123.013,223.315,-67.641,-178.816,9.613,149.573
C06104=1123.017,223.066,-67.615,-178.818,9.610,149.573
C06105=1123.021,222.817,-67.588,-178.821,9.607,149.573
C06106=1123.026,222.569,-67.562,-178.823,9.603,149.572
C06107=1123.030,222.320,-67.536,-178.826,9.600,149.572
C06108=1123.035,222.071,-67.510,-178.829,9.596,149.572
C06109=1123.039,221.823,-67.483,-178.832,9.594,149.572
C06110=1123.043,221.574,-67.457,-178.834,9.591,149.572
C06111=1123.047,221.326,-67.430,-178.837,9.587,149.572
C06112=1123.052,221.077,-67.405,-178.839,9.584,149.572
C06113=1123.056,220.829,-67.378,-178.841,9.581,149.572
C06114=1123.061,220.580,-67.352,-178.844,9.578,149.572
C06115=1123.065,220.332,-67.326,-178.846,9.575,149.572
C06116=1123.070,220.083,-67.299,-178.849,9.572,149.572
C06117=1123.074,219.834,-67.274,-178.852,9.568,149.572
C06118=1123.078,219.586,-67.247,-178.854,9.565,149.572
C06119=1123.083,219.337,-67.221,-178.857,9.562,149.572
C06120=1123.087,219.089,-67.194,-178.859,9.559,149.572
C06121=1123.091,218.840,-67.169,-178.861,9.556,149.571
C06122=1123.096,218.591,-67.142,-178.863,9.553,149.571
C06123=1123.101,218.343,-67.116,-178.866,9.550,149.571
C06124=1123.105,218.095,-67.090,-178.868,9.547,149.571
C06125=1123.109,217.846,-67.065,-178.870,9.544,149.571
C06126=1123.114,217.597,-67.038,-178.872,9.541,149.571
C06127=1123.118,217.349,-67.012,-178.875,9.538,149.571
C06128=1123.122,217.100,-66.986,-178.877,9.535,149.571
C06129=1123.127,216.852,-66.961,-178.879,9.532,149.570
C06130=1123.132,216.602,-66.934,-178.881,9.529,149.570
C06131=1123.136,216.354,-66.908,-178.884,9.526,149.570
C06132=1123.140,216.105,-66.882,-178.885,9.523,149.570
C06133=1123.144,215.857,-66.856,-178.888,9.520,149.570
C06134=1123.149,215.608,-66.831,-178.890,9.518,149.570
C06135=1123.154,215.359,-66.805,-178.892,9.515,149.570
C06136=1123.158,215.111,-66.778,-178.894,9.512,149.570
C06137=1123.162,214.862,-66.752,-178.896,9.509,149.570
C06138=1123.167,214.614,-66.727,-178.898,9.506,149.569
C06139=1123.171,214.365,-66.701,-178.900,9.503,149.569
C06140=1123.176,214.117,-66.676,-178.902,9.501,149.569
C06141=1123.181,213.868,-66.649,-178.904,9.498,149.569
C06142=1123.185,213.619,-66.623,-178.906,9.495,149.569
C06143=1123.189,213.370,-66.598,-178.908,9.492,149.569
C06144=1123.192,213.157,-66.576,-178.909,9.490,149.569
C06145=1123.197,212.942,-66.553,-178.911,9.488,149.569
C06146=1123.200,212.729,-66.531,-178.913,9.485,149.568
C06147=1123.204,212.515,-66.508,-178.915,9.483,149.568
C06148=1123.208,212.301,-66.487,-178.917,9.480,149.568
C06149=1123.212,212.088,-66.464,-178.918,9.478,149.568
C06150=1123.215,211.874,-66.443,-178.920,9.476,149.568
C06151=1123.219,211.660,-66.420,-178.922,9.473,149.568
C06152=1123.224,211.412,-66.395,-178.924,9.471,149.568
C06153=1123.228,211.163,-66.369,-178.927,9.468,149.568
C06154=1123.233,210.915,-66.343,-178.929,9.466,149.568
C06155=1123.238,210.666,-66.318,-178.931,9.463,149.568
C06156=1123.242,210.417,-66.293,-178.933,9.460,149.568
C06157=1123.246,210.168,-66.267,-178.936,9.457,149.568
C06158=1123.250,209.919,-66.241,-178.938,9.454,149.568
C06159=1123.255,209.671,-66.216,-178.940,9.452,149.568
C06160=1123.259,209.422,-66.190,-178.943,9.449,149.568
C06161=1123.264,209.174,-66.164,-178.945,9.446,149.568
C06162=1123.269,208.926,-66.139,-178.948,9.444,149.568
C06163=1123.273,208.677,-66.113,-178.950,9.441,149.568
C06164=1123.277,208.428,-66.087,-178.953,9.438,149.568
C06165=1123.282,208.179,-66.063,-178.955,9.436,149.568
C06166=1123.286,207.930,-66.037,-178.958,9.433,149.568
C06167=1123.291,207.682,-66.011,-178.961,9.430,149.568
C06168=1123.295,207.434,-65.986,-178.963,9.427,149.568
C06169=1123.300,207.185,-65.960,-178.966,9.424,149.568
C06170=1123.305,206.936,-65.935,-178.969,9.421,149.568
C06171=1123.309,206.687,-65.910,-178.971,9.419,149.568
C06172=1123.313,206.438,-65.884,-178.974,9.416,149.568
C06173=1123.318,206.190,-65.858,-178.976,9.413,149.568
C06174=1123.323,205.941,-65.833,-178.979,9.410,149.569
C06175=1123.327,205.692,-65.808,-178.982,9.408,149.569
C06176=1123.331,205.444,-65.783,-178.985,9.405,149.569
C06177=1123.335,205.195,-65.757,-178.988,9.402,149.569
C06178=1123.340,204.947,-65.732,-178.991,9.399,149.569
C06179=1123.344,204.698,-65.707,-178.994,9.396,149.569
C06180=1123.350,204.449,-65.682,-178.997,9.392,149.569
C06181=1123.354,204.200,-65.656,-179.000,9.390,149.569
C06182=1123.358,203.952,-65.631,-179.003,9.387,149.569
C06183=1123.362,203.703,-65.606,-179.006,9.384,149.569
C06184=1123.367,203.454,-65.581,-179.009,9.381,149.570
C06185=1123.372,203.206,-65.556,-179.012,9.379,149.570
C06186=1123.376,202.957,-65.530,-179.015,9.375,149.570
C06187=1123.381,202.709,-65.505,-179.018,9.372,149.570
C06188=1123.385,202.460,-65.480,-179.021,9.369,149.570
C06189=1123.389,202.212,-65.455,-179.024,9.366,149.570
C06190=1123.394,201.962,-65.430,-179.027,9.363,149.570
C06191=1123.399,201.714,-65.405,-179.030,9.360,149.570
C06192=1123.403,201.465,-65.380,-179.034,9.357,149.571
C06193=1123.407,201.217,-65.355,-179.036,9.354,149.570
C06194=1123.412,200.967,-65.330,-179.040,9.350,149.571
C06195=1123.416,200.719,-65.306,-179.043,9.347,149.571
C06196=1123.421,200.470,-65.280,-179.046,9.344,149.571
C06197=1123.426,200.221,-65.255,-179.050,9.340,149.571
C06198=1123.429,199.973,-65.230,-179.053,9.338,149.571
C06199=1123.434,199.724,-65.206,-179.056,9.334,149.571
C06200=1123.438,199.510,-65.184,-179.059,9.331,149.571
C06201=1123.442,199.296,-65.163,-179.062,9.328,149.571
C06202=1123.445,199.082,-65.141,-179.065,9.326,149.572
C06203=1123.450,198.868,-65.121,-179.068,9.323,149.572
C06204=1123.453,198.654,-65.099,-179.070,9.320,149.572
C06205=1123.458,198.440,-65.077,-179.073,9.317,149.572
C06206=1123.461,198.226,-65.056,-179.076,9.314,149.572
C06207=1123.465,198.013,-65.035,-179.079,9.310,149.572
C06208=1123.469,197.764,-65.010,-179.083,9.307,149.572
C06209=1123.474,197.515,-64.985,-179.086,9.304,149.572
C06210=1123.478,197.266,-64.961,-179.090,9.301,149.572
C06211=1123.483,197.018,-64.936,-179.093,9.297,149.572
C06212=1123.487,196.770,-64.912,-179.096,9.293,149.572
C06213=1123.492,196.520,-64.886,-179.101,9.289,149.573
C06214=1123.496,196.272,-64.862,-179.103,9.286,149.573
C06215=1123.501,196.022,-64.837,-179.105,9.283,149.572
C06216=1123.505,195.774,-64.813,-179.106,9.281,149.572
C06217=1123.510,195.525,-64.789,-179.108,9.278,149.572
C06218=1123.514,195.277,-64.763,-179.110,9.275,149.572
C06219=1123.519,195.028,-64.739,-179.112,9.273,149.572
C06220=1123.523,194.780,-64.715,-179.114,9.270,149.572
C06221=1123.528,194.530,-64.690,-179.116,9.268,149.572
C06222=1123.532,194.282,-64.666,-179.117,9.265,149.571
C06223=1123.537,194.033,-64.641,-179.119,9.263,149.571
C06224=1123.541,193.784,-64.617,-179.120,9.260,149.571
C06225=1123.546,193.535,-64.592,-179.123,9.257,149.571
C06226=1123.551,193.287,-64.568,-179.125,9.254,149.571
C06227=1123.555,193.038,-64.543,-179.126,9.252,149.571
C06228=1123.560,192.789,-64.519,-179.128,9.249,149.571
C06229=1123.564,192.540,-64.495,-179.131,9.246,149.571
C06230=1123.569,192.292,-64.470,-179.132,9.244,149.570
C06231=1123.573,192.043,-64.445,-179.134,9.241,149.570
C06232=1123.578,191.794,-64.421,-179.137,9.238,149.570
C06233=1123.583,191.545,-64.397,-179.139,9.236,149.570
C06234=1123.586,191.296,-64.372,-179.140,9.233,149.570
C06235=1123.591,191.048,-64.348,-179.143,9.230,149.570
C06236=1123.596,190.799,-64.324,-179.144,9.228,149.570
C06237=1123.601,190.550,-64.300,-179.147,9.225,149.570
C06238=1123.605,190.301,-64.275,-179.149,9.222,149.570
C06239=1123.609,190.052,-64.251,-179.151,9.220,149.570
C06240=1123.614,189.804,-64.227,-179.153,9.217,149.570
C06241=1123.619,189.555,-64.202,-179.155,9.214,149.570
C06242=1123.623,189.306,-64.178,-179.158,9.211,149.570
C06243=1123.627,189.057,-64.155,-179.160,9.208,149.570
C06244=1123.633,188.808,-64.130,-179.162,9.206,149.570
C06245=1123.637,188.560,-64.106,-179.165,9.203,149.570
C06246=1123.641,188.311,-64.081,-179.167,9.200,149.570
C06247=1123.646,188.062,-64.057,-179.169,9.197,149.570
C06248=1123.651,187.813,-64.033,-179.172,9.194,149.570
C06249=1123.655,187.565,-64.009,-179.173,9.192,149.569
C06250=1123.659,187.316,-63.985,-179.176,9.189,149.569
C06251=1123.664,187.067,-63.960,-179.179,9.186,149.569
C06252=1123.669,186.818,-63.937,-179.180,9.183,149.569
C06253=1123.673,186.569,-63.913,-179.183,9.180,149.569
C06254=1123.677,186.321,-63.889,-179.185,9.177,149.569
C06255=1123.683,186.072,-63.865,-179.188,9.174,149.569
C06256=1123.686,185.858,-63.844,-179.190,9.172,149.569
C06257=1123.690,185.644,-63.823,-179.192,9.169,149.569
C06258=1123.694,185.430,-63.803,-179.195,9.167,149.569
C06259=1123.698,185.216,-63.781,-179.197,9.164,149.569
C06260=1123.702,185.002,-63.761,-179.199,9.162,149.569
C06261=1123.705,184.787,-63.741,-179.201,9.159,149.569
C06262=1123.710,184.574,-63.720,-179.203,9.157,149.569
C06263=1123.713,184.360,-63.699,-179.205,9.154,149.569
C06264=1123.718,184.111,-63.675,-179.207,9.151,149.569
C06265=1123.723,183.862,-63.651,-179.210,9.148,149.569
C06266=1123.727,183.613,-63.628,-179.213,9.145,149.569
C06267=1123.732,183.365,-63.604,-179.215,9.142,149.569
C06268=1123.736,183.116,-63.580,-179.218,9.139,149.569
C06269=1123.741,182.867,-63.556,-179.221,9.135,149.569
C06270=1123.745,182.617,-63.533,-179.224,9.132,149.569
C06271=1123.749,182.369,-63.509,-179.227,9.129,149.569
C06272=1123.754,182.120,-63.485,-179.229,9.126,149.569
C06273=1123.758,181.872,-63.461,-179.232,9.123,149.569
C06274=1123.763,181.623,-63.438,-179.234,9.120,149.569
C06275=1123.768,181.374,-63.413,-179.238,9.116,149.569
C06276=1123.773,181.125,-63.390,-179.240,9.113,149.569
C06277=1123.778,180.876,-63.366,-179.243,9.110,149.569
C06278=1123.782,180.627,-63.342,-179.245,9.107,149.569
C06279=1123.787,180.378,-63.319,-179.248,9.103,149.569
C06280=1123.791,180.130,-63.295,-179.251,9.101,149.569
C06281=1123.796,179.881,-63.272,-179.255,9.097,149.569
C06282=1123.801,179.632,-63.248,-179.257,9.094,149.569
C06283=1123.804,179.384,-63.225,-179.260,9.090,149.569
C06284=1123.808,179.134,-63.201,-179.262,9.087,149.569
C06285=1123.813,178.885,-63.178,-179.265,9.084,149.569
C06286=1123.817,178.637,-63.154,-179.267,9.081,149.569
C06287=1123.822,178.388,-63.130,-179.269,9.078,149.569
C06288=1123.827,178.139,-63.107,-179.271,9.075,149.569
C06289=1123.832,177.890,-63.083,-179.273,9.072,149.568
C06290=1123.836,177.641,-63.059,-179.275,9.069,149.568
C06291=1123.841,177.392,-63.036,-179.278,9.066,149.568
C06292=1123.845,177.143,-63.013,-179.279,9.064,149.568
C06293=1123.850,176.894,-62.989,-179.282,9.061,149.568
C06294=1123.855,176.646,-62.966,-179.284,9.057,149.568
C06295=1123.859,176.398,-62.943,-179.286,9.055,149.568
C06296=1123.864,176.149,-62.920,-179.288,9.052,149.568
C06297=1123.868,175.900,-62.896,-179.291,9.049,149.568
C06298=1123.873,175.650,-62.873,-179.293,9.046,149.568
C06299=1123.878,175.401,-62.849,-179.295,9.043,149.567
C06300=1123.882,175.152,-62.826,-179.297,9.040,149.567
C06301=1123.887,174.903,-62.803,-179.299,9.037,149.567
C06302=1123.891,174.655,-62.779,-179.301,9.034,149.567
C06303=1123.896,174.406,-62.756,-179.304,9.031,149.567
C06304=1123.900,174.157,-62.733,-179.306,9.028,149.567
C06305=1123.905,173.908,-62.709,-179.308,9.025,149.567
C06306=1123.910,173.659,-62.686,-179.310,9.022,149.567
C06307=1123.914,173.410,-62.663,-179.313,9.019,149.567
C06308=1123.918,173.161,-62.640,-179.315,9.016,149.567
C06309=1123.923,172.912,-62.616,-179.317,9.013,149.566
C06310=1123.928,172.664,-62.593,-179.319,9.010,149.566
C06311=1123.932,172.415,-62.571,-179.321,9.007,149.566
C06312=1123.936,172.201,-62.550,-179.323,9.004,149.566
C06313=1123.940,171.987,-62.531,-179.325,9.002,149.566
C06314=1123.945,171.773,-62.510,-179.327,8.999,149.566
C06315=1123.948,171.558,-62.491,-179.329,8.997,149.566
C06316=1123.952,171.344,-62.471,-179.331,8.993,149.566
C06317=1123.957,171.130,-62.451,-179.333,8.991,149.566
C06318=1123.960,170.915,-62.431,-179.335,8.989,149.566
C06319=1123.964,170.702,-62.411,-179.337,8.986,149.566
C06320=1123.969,170.453,-62.388,-179.339,8.983,149.566
C06321=1123.973,170.204,-62.365,-179.341,8.980,149.566
C06322=1123.978,169.956,-62.342,-179.344,8.977,149.565
C06323=1123.983,169.706,-62.320,-179.346,8.974,149.565
C06324=1123.987,169.457,-62.296,-179.348,8.971,149.565
C06325=1123.991,169.208,-62.274,-179.350,8.968,149.565
C06326=1123.996,168.959,-62.250,-179.353,8.965,149.565
C06327=1124.001,168.710,-62.227,-179.355,8.962,149.565
C06328=1124.005,168.462,-62.204,-179.357,8.958,149.565
C06329=1124.010,168.213,-62.182,-179.360,8.955,149.565
C06330=1124.014,167.964,-62.159,-179.362,8.953,149.565
C06331=1124.019,167.715,-62.136,-179.364,8.949,149.565
C06332=1124.024,167.467,-62.113,-179.366,8.946,149.565
C06333=1124.029,167.217,-62.091,-179.369,8.943,149.564
C06334=1124.033,166.968,-62.067,-179.371,8.940,149.564
C06335=1124.037,166.719,-62.044,-179.374,8.936,149.564
C06336=1124.042,166.470,-62.021,-179.376,8.933,149.564
C06337=1124.048,166.221,-61.999,-179.379,8.930,149.564
C06338=1124.052,165.973,-61.976,-179.380,8.927,149.564
C06339=1124.056,165.724,-61.953,-179.383,8.924,149.564
C06340=1124.061,165.474,-61.931,-179.385,8.921,149.564
C06341=1124.066,165.226,-61.908,-179.388,8.918,149.564
C06342=1124.070,164.977,-61.886,-179.390,8.915,149.564
C06343=1124.075,164.728,-61.862,-179.392,8.912,149.564
C06344=1124.079,164.480,-61.840,-179.395,8.908,149.563
C06345=1124.084,164.230,-61.817,-179.397,8.905,149.563
C06346=1124.088,163.981,-61.794,-179.399,8.902,149.563
C06347=1124.093,163.732,-61.772,-179.402,8.899,149.563
C06348=1124.098,163.484,-61.749,-179.404,8.895,149.563
C06349=1124.102,163.234,-61.727,-179.407,8.892,149.563
C06350=1124.107,162.985,-61.704,-179.409,8.889,149.563
C06351=1124.111,162.737,-61.682,-179.411,8.886,149.563
C06352=1124.116,162.488,-61.659,-179.414,8.882,149.563
C06353=1124.120,162.239,-61.636,-179.416,8.879,149.563
C06354=1124.126,161.990,-61.614,-179.418,8.876,149.562
C06355=1124.130,161.741,-61.592,-179.421,8.873,149.562
C06356=1124.134,161.492,-61.569,-179.423,8.870,149.562
C06357=1124.140,161.243,-61.547,-179.425,8.866,149.562
C06358=1124.144,160.994,-61.524,-179.428,8.863,149.562
C06359=1124.148,160.745,-61.502,-179.430,8.860,149.562
C06360=1124.153,160.497,-61.479,-179.433,8.856,149.562
C06361=1124.158,160.247,-61.457,-179.435,8.853,149.562
C06362=1124.162,159.998,-61.435,-179.438,8.850,149.562
C06363=1124.167,159.749,-61.412,-179.440,8.847,149.561
C06364=1124.171,159.500,-61.390,-179.443,8.843,149.561
C06365=1124.176,159.252,-61.368,-179.445,8.840,149.561
C06366=1124.181,159.002,-61.345,-179.447,8.836,149.561
C06367=1124.185,158.753,-61.323,-179.450,8.833,149.561
C06368=1124.189,158.539,-61.304,-179.451,8.830,149.561
C06369=1124.193,158.325,-61.285,-179.454,8.827,149.561
C06370=1124.198,158.111,-61.266,-179.456,8.824,149.561
C06371=1124.202,157.896,-61.246,-179.458,8.822,149.561
C06372=1124.206,157.682,-61.227,-179.460,8.818,149.561
C06373=1124.210,157.468,-61.208,-179.462,8.816,149.561
C06374=1124.214,157.254,-61.189,-179.464,8.813,149.560
C06375=1124.217,157.039,-61.170,-179.467,8.810,149.560
C06376=1124.222,156.790,-61.148,-179.469,8.806,149.560
C06377=1124.226,156.542,-61.125,-179.472,8.803,149.560
C06378=1124.231,156.293,-61.104,-179.474,8.799,149.560
C06379=1124.236,156.043,-61.081,-179.476,8.796,149.560
C06380=1124.241,155.795,-61.059,-179.479,8.792,149.560
C06381=1124.245,155.545,-61.037,-179.481,8.789,149.559
C06382=1124.250,155.297,-61.016,-179.484,8.786,149.559
C06383=1124.254,155.047,-60.994,-179.486,8.782,149.559
C06384=1124.259,154.799,-60.972,-179.489,8.778,149.559
C06385=1124.264,154.550,-60.948,-179.491,8.775,149.559
C06386=1124.269,154.301,-60.927,-179.494,8.772,149.559
C06387=1124.273,154.052,-60.905,-179.496,8.768,149.559
C06388=1124.278,153.803,-60.883,-179.499,8.764,149.558
C06389=1124.282,153.554,-60.861,-179.501,8.761,149.558
C06390=1124.287,153.305,-60.839,-179.503,8.758,149.558
C06391=1124.291,153.056,-60.817,-179.506,8.754,149.558
C06392=1124.296,152.807,-60.796,-179.508,8.750,149.558
C06393=1124.301,152.557,-60.773,-179.511,8.747,149.558
C06394=1124.306,152.309,-60.751,-179.514,8.743,149.558
C06395=1124.311,152.060,-60.730,-179.516,8.740,149.558
C06396=1124.315,151.811,-60.708,-179.518,8.736,149.557
C06397=1124.320,151.562,-60.687,-179.521,8.732,149.557
C06398=1124.325,151.312,-60.665,-179.523,8.729,149.557
C06399=1124.330,151.064,-60.643,-179.526,8.725,149.557
C06400=1124.334,150.815,-60.621,-179.528,8.721,149.557
C06401=1124.339,150.566,-60.599,-179.531,8.718,149.557
C06402=1124.344,150.317,-60.577,-179.533,8.714,149.556
C06403=1124.348,150.068,-60.555,-179.536,8.710,149.556
C06404=1124.353,149.818,-60.534,-179.539,8.706,149.556
C06405=1124.358,149.570,-60.513,-179.541,8.703,149.556
C06406=1124.362,149.320,-60.491,-179.543,8.699,149.556
C06407=1124.367,149.072,-60.469,-179.546,8.695,149.556
C06408=1124.371,148.822,-60.447,-179.549,8.691,149.555
C06409=1124.376,148.573,-60.426,-179.551,8.688,149.555
C06410=1124.381,148.325,-60.405,-179.554,8.683,149.555
C06411=1124.385,148.075,-60.383,-179.556,8.680,149.555
C06412=1124.390,147.826,-60.362,-179.559,8.676,149.555
C06413=1124.395,147.578,-60.340,-179.561,8.673,149.554
C06414=1124.399,147.328,-60.318,-179.564,8.668,149.554
C06415=1124.404,147.080,-60.296,-179.566,8.665,149.554
C06416=1124.409,146.830,-60.276,-179.569,8.661,149.554
C06417=1124.414,146.582,-60.254,-179.571,8.657,149.554
C06418=1124.418,146.332,-60.233,-179.574,8.653,149.553
C06419=1124.423,146.083,-60.211,-179.576,8.649,149.553
C06420=1124.428,145.835,-60.190,-179.578,8.645,149.553
C06421=1124.432,145.585,-60.168,-179.581,8.642,149.553
C06422=1124.437,145.336,-60.147,-179.584,8.637,149.553
C06423=1124.442,145.087,-60.126,-179.586,8.634,149.552
C06424=1124.446,144.873,-60.107,-179.587,8.631,149.552
C06425=1124.450,144.658,-60.089,-179.589,8.628,149.552
C06426=1124.454,144.444,-60.071,-179.590,8.625,149.552
C06427=1124.458,144.229,-60.052,-179.591,8.622,149.551
C06428=1124.461,144.015,-60.034,-179.593,8.619,149.551
C06429=1124.466,143.801,-60.016,-179.594,8.616,149.551
C06430=1124.470,143.587,-59.998,-179.595,8.614,149.550
C06431=1124.474,143.372,-59.979,-179.597,8.611,149.550
C06432=1124.479,143.124,-59.958,-179.598,8.607,149.550
C06433=1124.483,142.874,-59.937,-179.599,8.604,149.549
C06434=1124.488,142.625,-59.915,-179.601,8.601,149.549
C06435=1124.493,142.376,-59.894,-179.602,8.597,149.549
C06436=1124.498,142.127,-59.873,-179.604,8.594,149.548
C06437=1124.502,141.878,-59.852,-179.605,8.591,149.548
C06438=1124.507,141.628,-59.831,-179.607,8.587,149.548
C06439=1124.512,141.380,-59.809,-179.608,8.584,149.547
C06440=1124.516,141.131,-59.789,-179.611,8.581,149.547
C06441=1124.521,140.882,-59.768,-179.612,8.578,149.547
C06442=1124.525,140.632,-59.746,-179.613,8.574,149.546
C06443=1124.530,140.383,-59.725,-179.615,8.571,149.546
C06444=1124.535,140.134,-59.705,-179.616,8.567,149.545
C06445=1124.540,139.885,-59.683,-179.618,8.564,149.545
C06446=1124.544,139.636,-59.662,-179.620,8.561,149.545
C06447=1124.550,139.387,-59.641,-179.621,8.557,149.545
C06448=1124.553,139.138,-59.620,-179.623,8.554,149.544
C06449=1124.558,138.889,-59.599,-179.625,8.551,149.544
C06450=1124.563,138.640,-59.578,-179.626,8.548,149.544
C06451=1124.568,138.391,-59.557,-179.628,8.544,149.543
C06452=1124.573,138.142,-59.536,-179.629,8.541,149.543
C06453=1124.577,137.893,-59.516,-179.631,8.537,149.543
C06454=1124.582,137.644,-59.495,-179.632,8.535,149.542
C06455=1124.587,137.395,-59.473,-179.634,8.531,149.542
C06456=1124.591,137.146,-59.452,-179.635,8.528,149.542
C06457=1124.596,136.896,-59.431,-179.637,8.525,149.541
C06458=1124.601,136.647,-59.411,-179.639,8.521,149.541
C06459=1124.606,136.398,-59.390,-179.640,8.518,149.541
C06460=1124.610,136.150,-59.369,-179.642,8.514,149.540
C06461=1124.615,135.901,-59.348,-179.643,8.511,149.540
C06462=1124.620,135.652,-59.328,-179.646,8.508,149.540
C06463=1124.624,135.402,-59.306,-179.647,8.505,149.539
C06464=1124.629,135.152,-59.285,-179.649,8.501,149.539
C06465=1124.634,134.903,-59.265,-179.650,8.498,149.539
C06466=1124.639,134.654,-59.244,-179.652,8.495,149.539
C06467=1124.643,134.406,-59.223,-179.654,8.491,149.538
C06468=1124.648,134.157,-59.202,-179.655,8.488,149.538
C06469=1124.653,133.908,-59.181,-179.657,8.485,149.538
C06470=1124.657,133.659,-59.161,-179.658,8.482,149.537
C06471=1124.662,133.409,-59.140,-179.660,8.478,149.537
C06472=1124.667,133.160,-59.120,-179.662,8.475,149.537
C06473=1124.672,132.911,-59.099,-179.663,8.472,149.537
C06474=1124.676,132.662,-59.078,-179.665,8.468,149.536
C06475=1124.682,132.413,-59.057,-179.667,8.465,149.536
C06476=1124.686,132.164,-59.037,-179.669,8.462,149.536
C06477=1124.691,131.915,-59.016,-179.670,8.458,149.535
C06478=1124.696,131.666,-58.996,-179.672,8.455,149.535
C06479=1124.700,131.417,-58.975,-179.674,8.452,149.535
C06480=1124.704,131.202,-58.957,-179.675,8.449,149.535
C06481=1124.708,130.988,-58.939,-179.677,8.446,149.534
C06482=1124.713,130.773,-58.923,-179.678,8.443,149.534
C06483=1124.716,130.559,-58.905,-179.679,8.441,149.534
C06484=1124.721,130.344,-58.886,-179.681,8.437,149.534
C06485=1124.725,130.130,-58.869,-179.683,8.434,149.533
C06486=1124.729,129.916,-58.851,-179.684,8.432,149.533
C06487=1124.732,129.701,-58.833,-179.685,8.429,149.533
C06488=1124.737,129.452,-58.812,-179.688,8.425,149.533
C06489=1124.742,129.202,-58.793,-179.689,8.422,149.532
C06490=1124.747,128.953,-58.772,-179.691,8.419,149.532
C06491=1124.752,128.704,-58.751,-179.692,8.416,149.532
C06492=1124.756,128.455,-58.731,-179.694,8.413,149.532
C06493=1124.761,128.206,-58.711,-179.696,8.409,149.531
C06494=1124.766,127.957,-58.690,-179.697,8.406,149.531
C06495=1124.771,127.707,-58.670,-179.699,8.403,149.531
C06496=1124.776,127.459,-58.650,-179.701,8.399,149.530
C06497=1124.781,127.210,-58.629,-179.702,8.396,149.530
C06498=1124.785,126.961,-58.609,-179.704,8.392,149.530
C06499=1124.790,126.712,-58.588,-179.706,8.389,149.530
C06500=1124.794,126.462,-58.569,-179.708,8.386,149.529
C06501=1124.800,126.213,-58.548,-179.710,8.382,149.529
C06502=1124.804,125.964,-58.527,-179.712,8.379,149.529
C06503=1124.808,125.715,-58.507,-179.714,8.375,149.528
C06504=1124.813,125.466,-58.487,-179.715,8.373,149.528
C06505=1124.818,125.217,-58.467,-179.717,8.369,149.528
C06506=1124.823,124.967,-58.446,-179.719,8.365,149.528
C06507=1124.828,124.718,-58.426,-179.720,8.363,149.527
C06508=1124.832,124.469,-58.406,-179.722,8.359,149.527
C06509=1124.837,124.221,-58.386,-179.724,8.355,149.527
C06510=1124.842,123.971,-58.366,-179.725,8.352,149.526
C06511=1124.847,123.722,-58.345,-179.727,8.349,149.526
C06512=1124.851,123.473,-58.325,-179.730,8.345,149.526
C06513=1124.856,123.223,-58.305,-179.732,8.342,149.526
C06514=1124.861,122.974,-58.285,-179.733,8.339,149.525
C06515=1124.865,122.725,-58.265,-179.735,8.335,149.525
C06516=1124.870,122.477,-58.245,-179.737,8.332,149.525
C06517=1124.875,122.228,-58.225,-179.739,8.328,149.525
C06518=1124.880,121.978,-58.205,-179.740,8.326,149.524
C06519=1124.885,121.729,-58.184,-179.742,8.322,149.524
C06520=1124.889,121.479,-58.165,-179.744,8.318,149.524
C06521=1124.894,121.230,-58.144,-179.746,8.315,149.524
C06522=1124.899,120.981,-58.125,-179.747,8.312,149.523
C06523=1124.904,120.732,-58.105,-179.749,8.309,149.523
C06524=1124.908,120.483,-58.085,-179.751,8.305,149.523
C06525=1124.913,120.234,-58.065,-179.753,8.301,149.522
C06526=1124.918,119.984,-58.045,-179.755,8.298,149.522
C06527=1124.922,119.735,-58.025,-179.757,8.295,149.522
C06528=1124.927,119.486,-58.005,-179.758,8.291,149.522
C06529=1124.932,119.238,-57.985,-179.760,8.288,149.521
C06530=1124.937,118.988,-57.965,-179.762,8.284,149.521
C06531=1124.941,118.738,-57.946,-179.764,8.281,149.521
C06532=1124.946,118.490,-57.926,-179.766,8.278,149.521
C06533=1124.951,118.241,-57.906,-179.768,8.274,149.520
C06534=1124.955,117.992,-57.886,-179.770,8.271,149.520
C06535=1124.960,117.742,-57.866,-179.772,8.267,149.520
C06536=1124.965,117.528,-57.849,-179.773,8.264,149.520
C06537=1124.968,117.313,-57.831,-179.775,8.262,149.519
C06538=1124.973,117.099,-57.815,-179.777,8.258,149.519
C06539=1124.977,116.884,-57.798,-179.778,8.255,149.519
C06540=1124.982,116.669,-57.781,-179.780,8.253,149.519
C06541=1124.985,116.455,-57.763,-179.781,8.250,149.518
C06542=1124.990,116.240,-57.747,-179.783,8.246,149.518
C06543=1124.994,116.025,-57.729,-179.784,8.244,149.518
C06544=1124.999,115.776,-57.710,-179.787,8.240,149.518
C06545=1125.003,115.527,-57.690,-179.788,8.236,149.517
C06546=1125.007,115.278,-57.671,-179.790,8.233,149.517
C06547=1125.013,115.029,-57.651,-179.792,8.229,149.517
C06548=1125.018,114.780,-57.632,-179.794,8.227,149.517
C06549=1125.022,114.531,-57.611,-179.795,8.223,149.516
C06550=1125.027,114.282,-57.592,-179.797,8.219,149.516
C06551=1125.032,114.032,-57.572,-179.799,8.216,149.516
C06552=1125.037,113.783,-57.553,-179.801,8.212,149.516
C06553=1125.042,113.534,-57.534,-179.804,8.209,149.515
C06554=1125.047,113.285,-57.513,-179.805,8.205,149.515
C06555=1125.051,113.036,-57.494,-179.807,8.201,149.515
C06556=1125.056,112.787,-57.475,-179.809,8.198,149.515
C06557=1125.061,112.537,-57.455,-179.811,8.194,149.514
C06558=1125.065,112.288,-57.435,-179.812,8.191,149.514
C06559=1125.071,112.039,-57.416,-179.814,8.188,149.514
C06560=1125.076,111.789,-57.397,-179.816,8.184,149.513
C06561=1125.080,111.540,-57.377,-179.819,8.181,149.513
C06562=1125.085,111.291,-57.358,-179.820,8.177,149.513
C06563=1125.089,111.042,-57.338,-179.822,8.173,149.513
C06564=1125.095,110.793,-57.319,-179.824,8.170,149.512
C06565=1125.099,110.544,-57.299,-179.827,8.166,149.512
C06566=1125.103,110.294,-57.280,-179.829,8.162,149.512
C06567=1125.109,110.046,-57.261,-179.832,8.158,149.512
C06568=1125.113,109.796,-57.241,-179.834,8.154,149.511
C06569=1125.118,109.547,-57.222,-179.837,8.150,149.511
C06570=1125.123,109.298,-57.202,-179.840,8.146,149.511
C06571=1125.128,109.048,-57.184,-179.842,8.143,149.511
C06572=1125.133,108.799,-57.164,-179.844,8.138,149.511
C06573=1125.137,108.550,-57.145,-179.846,8.134,149.510
C06574=1125.143,108.301,-57.126,-179.849,8.130,149.510
C06575=1125.147,108.051,-57.106,-179.851,8.127,149.510
C06576=1125.152,107.803,-57.088,-179.853,8.123,149.510
C06577=1125.157,107.553,-57.068,-179.855,8.119,149.509
C06578=1125.162,107.304,-57.049,-179.857,8.115,149.509
C06579=1125.166,107.055,-57.030,-179.860,8.111,149.509
C06580=1125.172,106.805,-57.011,-179.862,8.108,149.509
C06581=1125.176,106.556,-56.992,-179.865,8.103,149.509
C06582=1125.181,106.307,-56.973,-179.867,8.099,149.508
C06583=1125.186,106.058,-56.953,-179.869,8.095,149.508
C06584=1125.190,105.809,-56.934,-179.871,8.092,149.508
C06585=1125.195,105.559,-56.915,-179.873,8.088,149.507
C06586=1125.200,105.310,-56.897,-179.876,8.084,149.507
C06587=1125.205,105.061,-56.877,-179.878,8.080,149.507
C06588=1125.210,104.812,-56.859,-179.880,8.076,149.507
C06589=1125.214,104.562,-56.839,-179.882,8.072,149.506
C06590=1125.220,104.313,-56.820,-179.884,8.068,149.506
C06591=1125.224,104.064,-56.801,-179.887,8.064,149.506
C06592=1125.229,103.849,-56.785,-179.889,8.061,149.506
C06593=1125.232,103.635,-56.769,-179.890,8.057,149.505
C06594=1125.237,103.420,-56.752,-179.892,8.054,149.505
C06595=1125.241,103.205,-56.736,-179.894,8.050,149.505
C06596=1125.245,102.991,-56.720,-179.896,8.047,149.504
C06597=1125.249,102.776,-56.704,-179.897,8.044,149.504
C06598=1125.254,102.561,-56.688,-179.899,8.040,149.504
C06599=1125.257,102.347,-56.671,-179.901,8.037,149.504
C06600=1125.263,102.097,-56.653,-179.903,8.033,149.503
C06601=1125.267,101.849,-56.634,-179.905,8.029,149.503
C06602=1125.272,101.599,-56.614,-179.907,8.025,149.503
C06603=1125.277,101.350,-56.596,-179.909,8.021,149.502
C06604=1125.281,101.101,-56.577,-179.910,8.017,149.502
C06605=1125.287,100.851,-56.559,-179.913,8.013,149.502
C06606=1125.291,100.603,-56.540,-179.915,8.009,149.501
C06607=1125.296,100.352,-56.521,-179.917,8.006,149.501
C06608=1125.301,100.104,-56.502,-179.918,8.002,149.501
C06609=1125.306,99.855,-56.484,-179.921,7.997,149.500
C06610=1125.311,99.604,-56.465,-179.923,7.994,149.500
C06611=1125.315,99.356,-56.447,-179.924,7.990,149.499
C06612=1125.320,99.107,-56.429,-179.926,7.986,149.499
C06613=1125.325,98.857,-56.409,-179.929,7.982,149.499
C06614=1125.330,98.608,-56.391,-179.930,7.978,149.498
C06615=1125.335,98.359,-56.372,-179.932,7.974,149.498
C06616=1125.340,98.109,-56.353,-179.934,7.970,149.498
C06617=1125.345,97.860,-56.336,-179.935,7.966,149.497
C06618=1125.349,97.611,-56.317,-179.938,7.962,149.497
C06619=1125.354,97.361,-56.298,-179.939,7.958,149.496
C06620=1125.359,97.112,-56.280,-179.941,7.954,149.496
C06621=1125.364,96.864,-56.261,-179.943,7.950,149.496
C06622=1125.369,96.613,-56.242,-179.945,7.947,149.495
C06623=1125.374,96.364,-56.224,-179.946,7.943,149.495
C06624=1125.379,96.115,-56.206,-179.948,7.939,149.495
C06625=1125.383,95.866,-56.188,-179.950,7.934,149.494
C06626=1125.388,95.616,-56.169,-179.952,7.931,149.494
C06627=1125.393,95.367,-56.151,-179.954,7.927,149.493
C06628=1125.398,95.118,-56.133,-179.955,7.923,149.493
C06629=1125.403,94.869,-56.114,-179.957,7.919,149.493
C06630=1125.407,94.619,-56.096,-179.958,7.915,149.492
C06631=1125.413,94.370,-56.077,-179.960,7.911,149.492
C06632=1125.418,94.121,-56.059,-179.962,7.907,149.491
C06633=1125.422,93.872,-56.041,-179.963,7.903,149.491
C06634=1125.427,93.623,-56.022,-179.965,7.900,149.490
C06635=1125.431,93.373,-56.004,-179.966,7.896,149.490
C06636=1125.436,93.124,-55.986,-179.968,7.892,149.490
C06637=1125.442,92.875,-55.968,-179.970,7.888,149.489
C06638=1125.447,92.625,-55.950,-179.971,7.884,149.489
C06639=1125.452,92.376,-55.932,-179.973,7.880,149.488
C06640=1125.456,92.126,-55.913,-179.974,7.876,149.488
C06641=1125.461,91.877,-55.895,-179.976,7.872,149.487
C06642=1125.466,91.628,-55.877,-179.978,7.868,149.487
C06643=1125.471,91.379,-55.859,-179.979,7.865,149.487
C06644=1125.475,91.130,-55.841,-179.981,7.861,149.486
C06645=1125.480,90.880,-55.822,-179.982,7.857,149.486
C06646=1125.485,90.631,-55.804,-179.984,7.853,149.485
C06647=1125.490,90.382,-55.786,-179.985,7.849,149.485
C06648=1125.494,90.167,-55.770,-179.987,7.845,149.484
C06649=1125.499,89.952,-55.755,-179.988,7.842,149.484
C06650=1125.503,89.738,-55.740,-179.989,7.839,149.484
C06651=1125.507,89.523,-55.724,-179.991,7.835,149.483
C06652=1125.512,89.308,-55.708,-179.992,7.832,149.483
C06653=1125.516,89.093,-55.693,-179.993,7.828,149.482
C06654=1125.520,88.878,-55.677,-179.994,7.825,149.482
C06655=1125.524,88.664,-55.662,-179.995,7.822,149.481
C06656=1125.529,88.414,-55.644,-179.997,7.818,149.481
C06657=1125.534,88.165,-55.626,-179.998,7.814,149.481
C06658=1125.539,87.916,-55.608,180.000,7.810,149.480
C06659=1125.543,87.666,-55.590,179.998,7.806,149.480
C06660=1125.548,87.417,-55.572,179.998,7.803,149.479
C06661=1125.553,87.168,-55.554,179.996,7.799,149.479
C06662=1125.558,86.918,-55.537,179.995,7.795,149.478
C06663=1125.563,86.669,-55.519,179.993,7.791,149.478
C06664=1125.568,86.420,-55.501,179.992,7.787,149.477
C06665=1125.573,86.170,-55.483,179.990,7.783,149.477
C06666=1125.578,85.921,-55.465,179.989,7.780,149.476
C06667=1125.583,85.672,-55.447,179.988,7.775,149.476
C06668=1125.588,85.422,-55.429,179.987,7.771,149.475
C06669=1125.592,85.173,-55.412,179.985,7.768,149.475
C06670=1125.597,84.924,-55.394,179.985,7.764,149.474
C06671=1125.602,84.675,-55.376,179.983,7.760,149.474
C06672=1125.607,84.426,-55.358,179.981,7.756,149.473
C06673=1125.612,84.176,-55.341,179.980,7.752,149.473
C06674=1125.617,83.927,-55.323,179.979,7.749,149.472
C06675=1125.621,83.677,-55.304,179.978,7.745,149.472
C06676=1125.626,83.427,-55.287,179.977,7.741,149.471
C06677=1125.631,83.178,-55.269,179.976,7.738,149.471
C06678=1125.636,82.929,-55.252,179.974,7.733,149.470
C06679=1125.640,82.680,-55.234,179.973,7.729,149.470
C06680=1125.646,82.430,-55.217,179.972,7.726,149.469
C06681=1125.651,82.181,-55.199,179.971,7.722,149.469
C06682=1125.656,81.932,-55.181,179.970,7.718,149.468
C06683=1125.661,81.682,-55.163,179.969,7.715,149.468
C06684=1125.665,81.433,-55.146,179.968,7.710,149.467
C06685=1125.670,81.183,-55.129,179.967,7.707,149.466
C06686=1125.676,80.935,-55.111,179.965,7.703,149.466
C06687=1125.681,80.686,-55.093,179.964,7.699,149.465
C06688=1125.686,80.436,-55.076,179.963,7.696,149.465
C06689=1125.690,80.187,-55.058,179.962,7.692,149.464
C06690=1125.695,79.937,-55.041,179.961,7.689,149.464
C06691=1125.700,79.688,-55.023,179.960,7.684,149.463
C06692=1125.705,79.439,-55.005,179.959,7.681,149.463
C06693=1125.709,79.190,-54.989,179.958,7.677,149.462
C06694=1125.714,78.940,-54.971,179.957,7.673,149.462
C06695=1125.720,78.691,-54.953,179.956,7.669,149.461
C06696=1125.725,78.441,-54.935,179.955,7.666,149.460
C06697=1125.729,78.192,-54.919,179.953,7.662,149.460
C06698=1125.734,77.943,-54.901,179.953,7.659,149.459
C06699=1125.739,77.693,-54.883,179.951,7.655,149.459
C06700=1125.744,77.444,-54.865,179.951,7.651,149.458
C06701=1125.749,77.194,-54.849,179.950,7.647,149.458
C06702=1125.754,76.946,-54.831,179.949,7.644,149.457
C06703=1125.759,76.696,-54.814,179.948,7.640,149.457
C06704=1125.763,76.481,-54.798,179.947,7.636,149.456
C06705=1125.767,76.266,-54.784,179.946,7.633,149.456
C06706=1125.771,76.052,-54.769,179.944,7.630,149.456
C06707=1125.776,75.836,-54.754,179.943,7.627,149.455
C06708=1125.780,75.621,-54.739,179.941,7.623,149.455
C06709=1125.784,75.407,-54.724,179.940,7.620,149.454
C06710=1125.789,75.192,-54.709,179.939,7.616,149.454
C06711=1125.792,74.978,-54.695,179.938,7.613,149.453
C06712=1125.798,74.728,-54.677,179.936,7.609,149.453
C06713=1125.803,74.478,-54.660,179.935,7.604,149.452
C06714=1125.807,74.229,-54.643,179.933,7.600,149.452
C06715=1125.812,73.979,-54.625,179.932,7.597,149.451
C06716=1125.817,73.730,-54.609,179.930,7.593,149.451
C06717=1125.822,73.481,-54.591,179.929,7.588,149.450
C06718=1125.827,73.232,-54.574,179.928,7.584,149.450
C06719=1125.832,72.982,-54.557,179.927,7.581,149.450
C06720=1125.837,72.733,-54.539,179.925,7.577,149.449
C06721=1125.841,72.484,-54.522,179.924,7.573,149.448
C06722=1125.847,72.234,-54.506,179.922,7.569,149.448
C06723=1125.852,71.985,-54.489,179.921,7.565,149.448
C06724=1125.856,71.736,-54.471,179.919,7.561,149.447
C06725=1125.862,71.486,-54.454,179.918,7.557,149.447
C06726=1125.866,71.236,-54.437,179.916,7.553,149.446
C06727=1125.872,70.987,-54.420,179.915,7.549,149.446
C06728=1125.876,70.739,-54.403,179.913,7.545,149.445
C06729=1125.881,70.489,-54.385,179.912,7.541,149.445
C06730=1125.886,70.239,-54.369,179.911,7.537,149.444
C06731=1125.891,69.989,-54.352,179.909,7.533,149.444
C06732=1125.896,69.741,-54.335,179.908,7.529,149.443
C06733=1125.901,69.491,-54.318,179.906,7.525,149.443
C06734=1125.906,69.241,-54.301,179.905,7.521,149.442
C06735=1125.911,68.992,-54.283,179.903,7.517,149.442
C06736=1125.916,68.743,-54.267,179.902,7.513,149.441
C06737=1125.920,68.494,-54.250,179.901,7.509,149.441
C06738=1125.926,68.244,-54.233,179.899,7.505,149.440
C06739=1125.930,67.995,-54.216,179.898,7.501,149.440
C06740=1125.936,67.746,-54.199,179.896,7.497,149.439
C06741=1125.940,67.496,-54.183,179.895,7.493,149.439
C06742=1125.946,67.246,-54.166,179.893,7.489,149.438
C06743=1125.951,66.998,-54.149,179.892,7.485,149.438
C06744=1125.955,66.748,-54.133,179.890,7.481,149.437
C06745=1125.960,66.498,-54.115,179.889,7.478,149.437
C06746=1125.965,66.249,-54.099,179.888,7.474,149.436
C06747=1125.970,66.000,-54.082,179.887,7.470,149.436
C06748=1125.975,65.750,-54.065,179.885,7.466,149.435
C06749=1125.980,65.501,-54.048,179.884,7.462,149.435
C06750=1125.985,65.252,-54.032,179.883,7.458,149.434
C06751=1125.990,65.002,-54.015,179.881,7.454,149.434
C06752=1125.994,64.753,-53.998,179.880,7.449,149.433
C06753=1125.999,64.504,-53.982,179.878,7.446,149.433
C06754=1126.005,64.254,-53.965,179.877,7.442,149.432
C06755=1126.009,64.005,-53.948,179.876,7.437,149.432
C06756=1126.014,63.756,-53.932,179.874,7.433,149.431
C06757=1126.019,63.506,-53.914,179.873,7.430,149.431
C06758=1126.024,63.256,-53.898,179.871,7.425,149.430
C06759=1126.029,63.007,-53.882,179.870,7.421,149.430
C06760=1126.034,62.792,-53.867,179.869,7.418,149.429
C06761=1126.037,62.577,-53.853,179.867,7.414,149.429
C06762=1126.042,62.362,-53.839,179.866,7.411,149.429
C06763=1126.046,62.147,-53.825,179.865,7.407,149.428
C06764=1126.051,61.932,-53.811,179.864,7.404,149.428
C06765=1126.055,61.717,-53.797,179.863,7.401,149.427
C06766=1126.059,61.502,-53.782,179.861,7.397,149.427
C06767=1126.064,61.288,-53.768,179.860,7.394,149.426
C06768=1126.068,61.038,-53.752,179.859,7.390,149.426
C06769=1126.073,60.788,-53.734,179.858,7.386,149.425
C06770=1126.078,60.540,-53.718,179.856,7.382,149.425
C06771=1126.083,60.289,-53.702,179.855,7.378,149.424
C06772=1126.088,60.041,-53.686,179.854,7.374,149.424
C06773=1126.093,59.791,-53.669,179.852,7.370,149.423
C06774=1126.099,59.542,-53.652,179.851,7.365,149.423
C06775=1126.103,59.292,-53.636,179.849,7.362,149.422
C06776=1126.108,59.043,-53.620,179.848,7.357,149.422
C06777=1126.113,58.794,-53.603,179.847,7.353,149.421
C06778=1126.118,58.544,-53.587,179.845,7.349,149.421
C06779=1126.123,58.295,-53.571,179.844,7.345,149.420
C06780=1126.127,58.045,-53.554,179.842,7.341,149.420
C06781=1126.133,57.796,-53.538,179.841,7.337,149.419
C06782=1126.138,57.546,-53.521,179.840,7.333,149.419
C06783=1126.143,57.297,-53.506,179.838,7.329,149.418
C06784=1126.148,57.047,-53.489,179.838,7.326,149.418
C06785=1126.153,56.799,-53.473,179.836,7.322,149.417
C06786=1126.158,56.548,-53.457,179.835,7.317,149.417
C06787=1126.163,56.300,-53.441,179.834,7.313,149.416
C06788=1126.167,56.050,-53.425,179.832,7.309,149.416
C06789=1126.173,55.801,-53.408,179.831,7.305,149.415
C06790=1126.177,55.551,-53.392,179.829,7.301,149.415
C06791=1126.182,55.302,-53.376,179.828,7.297,149.414
C06792=1126.187,55.052,-53.360,179.827,7.293,149.414
C06793=1126.192,54.803,-53.344,179.826,7.289,149.413
C06794=1126.198,54.553,-53.327,179.824,7.285,149.413
C06795=1126.203,54.304,-53.311,179.823,7.281,149.412
C06796=1126.208,54.054,-53.295,179.821,7.277,149.411
C06797=1126.213,53.805,-53.279,179.820,7.272,149.411
C06798=1126.218,53.555,-53.263,179.819,7.269,149.410
C06799=1126.223,53.306,-53.247,179.818,7.264,149.410
C06800=1126.228,53.057,-53.231,179.816,7.260,149.409
C06801=1126.232,52.807,-53.214,179.815,7.256,149.409
C06802=1126.238,52.558,-53.199,179.813,7.252,149.408
C06803=1126.242,52.309,-53.184,179.812,7.248,149.408
C06804=1126.247,52.059,-53.167,179.811,7.244,149.407
C06805=1126.252,51.810,-53.151,179.810,7.240,149.407
C06806=1126.257,51.560,-53.135,179.808,7.236,149.406
C06807=1126.262,51.311,-53.119,179.807,7.231,149.405
C06808=1126.268,51.061,-53.104,179.805,7.227,149.405
C06809=1126.272,50.811,-53.088,179.804,7.223,149.404
C06810=1126.277,50.563,-53.071,179.803,7.219,149.404
C06811=1126.282,50.312,-53.055,179.802,7.215,149.403
C06812=1126.288,50.063,-53.040,179.800,7.211,149.403
C06813=1126.293,49.814,-53.023,179.799,7.207,149.402
C06814=1126.298,49.564,-53.008,179.798,7.203,149.402
C06815=1126.302,49.315,-52.993,179.797,7.199,149.401
C06816=1126.307,49.100,-52.978,179.796,7.195,149.401
C06817=1126.311,48.885,-52.965,179.795,7.192,149.400
C06818=1126.315,48.670,-52.951,179.793,7.188,149.400
C06819=1126.319,48.455,-52.938,179.793,7.185,149.399
C06820=1126.324,48.240,-52.924,179.791,7.181,149.399
C06821=1126.328,48.025,-52.911,179.790,7.178,149.398
C06822=1126.333,47.810,-52.896,179.789,7.175,149.398
C06823=1126.337,47.594,-52.883,179.788,7.170,149.397
C06824=1126.341,47.345,-52.868,179.787,7.166,149.397
C06825=1126.347,47.096,-52.852,179.785,7.162,149.396
C06826=1126.351,46.847,-52.836,179.784,7.158,149.396
C06827=1126.357,46.597,-52.820,179.783,7.154,149.395
C06828=1126.362,46.348,-52.805,179.781,7.150,149.395
C06829=1126.366,46.098,-52.789,179.780,7.146,149.394
C06830=1126.372,45.849,-52.774,179.779,7.141,149.393
C06831=1126.377,45.599,-52.758,179.778,7.137,149.393
C06832=1126.382,45.350,-52.743,179.776,7.133,149.392
C06833=1126.386,45.100,-52.727,179.775,7.129,149.392
C06834=1126.392,44.851,-52.712,179.774,7.125,149.391
C06835=1126.397,44.602,-52.695,179.773,7.121,149.391
C06836=1126.402,44.352,-52.679,179.771,7.117,149.390
C06837=1126.406,44.103,-52.664,179.770,7.112,149.390
C06838=1126.412,43.853,-52.649,179.769,7.108,149.389
C06839=1126.417,43.604,-52.633,179.768,7.104,149.389
C06840=1126.421,43.354,-52.618,179.766,7.100,149.388
C06841=1126.426,43.105,-52.602,179.765,7.096,149.387
C06842=1126.432,42.855,-52.587,179.764,7.092,149.387
C06843=1126.437,42.606,-52.572,179.763,7.087,149.386
C06844=1126.442,42.357,-52.556,179.762,7.083,149.386
C06845=1126.447,42.107,-52.540,179.760,7.079,149.385
C06846=1126.452,41.857,-52.526,179.759,7.075,149.384
C06847=1126.457,41.607,-52.510,179.758,7.070,149.384
C06848=1126.462,41.358,-52.495,179.757,7.066,149.383
C06849=1126.467,41.109,-52.480,179.755,7.062,149.383
C06850=1126.472,40.859,-52.464,179.754,7.058,149.382
C06851=1126.477,40.609,-52.448,179.753,7.054,149.381
C06852=1126.482,40.360,-52.433,179.752,7.050,149.381
C06853=1126.487,40.111,-52.418,179.751,7.045,149.380
C06854=1126.492,39.862,-52.403,179.750,7.041,149.380
C06855=1126.498,39.612,-52.388,179.748,7.037,149.379
C06856=1126.502,39.362,-52.372,179.747,7.033,149.379
C06857=1126.507,39.113,-52.357,179.746,7.029,149.378
C06858=1126.512,38.863,-52.341,179.745,7.024,149.377
C06859=1126.517,38.614,-52.326,179.744,7.020,149.377
C06860=1126.522,38.365,-52.311,179.742,7.016,149.376
C06861=1126.527,38.115,-52.296,179.741,7.012,149.376
C06862=1126.533,37.866,-52.281,179.740,7.007,149.375
C06863=1126.537,37.616,-52.265,179.739,7.003,149.374
C06864=1126.542,37.366,-52.250,179.737,6.999,149.374
C06865=1126.547,37.117,-52.235,179.736,6.995,149.373
C06866=1126.553,36.867,-52.220,179.735,6.991,149.373
C06867=1126.557,36.618,-52.205,179.734,6.986,149.372
C06868=1126.563,36.369,-52.189,179.733,6.982,149.371
C06869=1126.568,36.119,-52.175,179.732,6.978,149.371
C06870=1126.573,35.870,-52.159,179.731,6.974,149.370
C06871=1126.578,35.621,-52.144,179.729,6.969,149.370
C06872=1126.582,35.405,-52.131,179.729,6.966,149.369
C06873=1126.587,35.189,-52.119,179.727,6.962,149.369
C06874=1126.591,34.974,-52.106,179.727,6.959,149.368
C06875=1126.596,34.759,-52.093,179.726,6.954,149.367
C06876=1126.600,34.544,-52.079,179.725,6.951,149.367
C06877=1126.604,34.329,-52.067,179.724,6.947,149.366
C06878=1126.608,34.114,-52.054,179.723,6.944,149.366
C06879=1126.613,33.899,-52.041,179.722,6.940,149.365
C06880=1126.617,33.650,-52.026,179.720,6.935,149.365
C06881=1126.623,33.400,-52.011,179.719,6.931,149.364
C06882=1126.628,33.151,-51.996,179.718,6.927,149.364
C06883=1126.633,32.900,-51.981,179.717,6.923,149.363
C06884=1126.638,32.651,-51.966,179.716,6.918,149.362
C06885=1126.643,32.402,-51.952,179.715,6.914,149.362
C06886=1126.648,32.152,-51.936,179.714,6.910,149.361
C06887=1126.653,31.902,-51.922,179.713,6.905,149.360
C06888=1126.657,31.653,-51.907,179.712,6.901,149.360
C06889=1126.663,31.403,-51.892,179.710,6.897,149.359
C06890=1126.668,31.154,-51.877,179.709,6.893,149.358
C06891=1126.673,30.904,-51.863,179.708,6.888,149.358
C06892=1126.678,30.655,-51.847,179.707,6.884,149.357
C06893=1126.683,30.405,-51.833,179.706,6.880,149.356
C06894=1126.688,30.156,-51.818,179.705,6.874,149.356
C06895=1126.693,29.906,-51.803,179.703,6.870,149.355
C06896=1126.699,29.658,-51.788,179.702,6.866,149.354
C06897=1126.704,29.408,-51.774,179.701,6.862,149.354
C06898=1126.709,29.158,-51.760,179.700,6.857,149.353
C06899=1126.714,28.909,-51.744,179.699,6.853,149.353
C06900=1126.719,28.659,-51.730,179.698,6.849,149.352
C06901=1126.724,28.410,-51.715,179.697,6.844,149.351
C06902=1126.729,28.161,-51.701,179.696,6.840,149.351
C06903=1126.734,27.911,-51.686,179.695,6.836,149.350
C06904=1126.739,27.661,-51.671,179.694,6.831,149.349
C06905=1126.744,27.412,-51.657,179.693,6.827,149.349
C06906=1126.749,27.162,-51.642,179.692,6.823,149.348
C06907=1126.754,26.913,-51.627,179.691,6.818,149.347
C06908=1126.759,26.663,-51.612,179.690,6.814,149.347
C06909=1126.764,26.413,-51.598,179.688,6.809,149.346
C06910=1126.770,26.164,-51.584,179.687,6.805,149.345
C06911=1126.774,25.915,-51.569,179.686,6.800,149.345
C06912=1126.779,25.665,-51.555,179.685,6.796,149.344
C06913=1126.785,25.415,-51.540,179.684,6.792,149.343
C06914=1126.790,25.166,-51.526,179.683,6.787,149.343
C06915=1126.795,24.917,-51.511,179.682,6.783,149.342
C06916=1126.800,24.667,-51.496,179.681,6.778,149.341
C06917=1126.804,24.417,-51.482,179.680,6.774,149.341
C06918=1126.810,24.168,-51.468,179.679,6.770,149.340
C06919=1126.815,23.918,-51.454,179.678,6.765,149.339
C06920=1126.820,23.669,-51.438,179.676,6.760,149.339
C06921=1126.825,23.419,-51.424,179.675,6.756,149.338
C06922=1126.830,23.170,-51.410,179.674,6.752,149.337
C06923=1126.835,22.920,-51.396,179.674,6.747,149.337
C06924=1126.841,22.671,-51.382,179.673,6.743,149.336
C06925=1126.846,22.421,-51.367,179.672,6.738,149.335
C06926=1126.851,22.171,-51.353,179.671,6.734,149.335
C06927=1126.856,21.922,-51.339,179.670,6.730,149.334
C06928=1126.860,21.707,-51.326,179.668,6.725,149.333
C06929=1126.864,21.492,-51.314,179.668,6.722,149.333
C06930=1126.869,21.277,-51.301,179.667,6.717,149.332
C06931=1126.873,21.061,-51.290,179.666,6.714,149.332
C06932=1126.878,20.846,-51.277,179.665,6.710,149.331
C06933=1126.882,20.631,-51.265,179.664,6.706,149.330
C06934=1126.887,20.415,-51.253,179.664,6.702,149.330
C06935=1126.891,20.201,-51.240,179.663,6.698,149.329
C06936=1126.896,19.951,-51.226,179.662,6.694,149.328
C06937=1126.901,19.701,-51.212,179.660,6.689,149.328
C06938=1126.906,19.452,-51.197,179.659,6.685,149.327
C06939=1126.911,19.202,-51.183,179.659,6.680,149.326
C06940=1126.916,18.953,-51.169,179.658,6.676,149.325
C06941=1126.921,18.703,-51.155,179.657,6.672,149.325
C06942=1126.926,18.454,-51.141,179.656,6.666,149.324
C06943=1126.932,18.204,-51.127,179.655,6.662,149.323
C06944=1126.937,17.954,-51.113,179.654,6.657,149.323
C06945=1126.942,17.705,-51.099,179.653,6.653,149.322
C06946=1126.947,17.455,-51.085,179.652,6.648,149.321
C06947=1126.952,17.206,-51.071,179.651,6.644,149.320
C06948=1126.957,16.956,-51.056,179.650,6.639,149.320
C06949=1126.962,16.707,-51.043,179.649,6.634,149.319
C06950=1126.966,16.457,-51.028,179.648,6.630,149.318
C06951=1126.972,16.208,-51.014,179.647,6.625,149.317
C06952=1126.977,15.958,-51.001,179.646,6.621,149.317
C06953=1126.982,15.708,-50.987,179.645,6.617,149.316
C06954=1126.988,15.459,-50.973,179.644,6.612,149.315
C06955=1126.993,15.209,-50.958,179.643,6.607,149.315
C06956=1126.998,14.960,-50.944,179.642,6.602,149.314
C06957=1127.003,14.710,-50.932,179.641,6.598,149.313
C06958=1127.008,14.460,-50.917,179.641,6.593,149.312
C06959=1127.013,14.211,-50.903,179.640,6.589,149.312
C06960=1127.018,13.962,-50.889,179.639,6.584,149.311
C06961=1127.024,13.711,-50.876,179.637,6.579,149.310
C06962=1127.028,13.462,-50.862,179.636,6.574,149.309
C06963=1127.033,13.213,-50.848,179.636,6.570,149.309
C06964=1127.038,12.963,-50.834,179.635,6.565,149.308
C06965=1127.044,12.714,-50.820,179.634,6.561,149.307
C06966=1127.049,12.464,-50.806,179.633,6.556,149.306
C06967=1127.053,12.215,-50.793,179.632,6.551,149.305
C06968=1127.059,11.965,-50.779,179.631,6.547,149.305
C06969=1127.064,11.715,-50.765,179.630,6.542,149.304
C06970=1127.070,11.466,-50.751,179.629,6.537,149.303
C06971=1127.074,11.216,-50.738,179.628,6.532,149.302
C06972=1127.079,10.966,-50.724,179.627,6.528,149.302
C06973=1127.085,10.717,-50.710,179.627,6.523,149.301
C06974=1127.090,10.467,-50.696,179.626,6.518,149.300
C06975=1127.095,10.218,-50.683,179.625,6.514,149.299
C06976=1127.100,9.968,-50.670,179.624,6.508,149.298
C06977=1127.105,9.718,-50.655,179.623,6.504,149.298
C06978=1127.110,9.470,-50.642,179.622,6.499,149.297
C06979=1127.115,9.219,-50.628,179.622,6.495,149.296
C06980=1127.121,8.970,-50.614,179.621,6.490,149.295
C06981=1127.125,8.720,-50.602,179.620,6.485,149.295
C06982=1127.131,8.471,-50.588,179.619,6.480,149.294
C06983=1127.136,8.221,-50.574,179.618,6.476,149.293
C06984=1127.140,8.006,-50.562,179.618,6.472,149.292
C06985=1127.144,7.790,-50.551,179.617,6.467,149.291
C06986=1127.149,7.576,-50.539,179.617,6.464,149.291
C06987=1127.154,7.360,-50.527,179.617,6.460,149.290
C06988=1127.158,7.145,-50.515,179.616,6.456,149.289
C06989=1127.163,6.929,-50.504,179.616,6.453,149.288
C06990=1127.167,6.714,-50.493,179.615,6.448,149.288
C06991=1127.171,6.499,-50.481,179.615,6.445,149.287
C06992=1127.177,6.250,-50.467,179.614,6.440,149.286
C06993=1127.181,6.000,-50.454,179.615,6.436,149.285
C06994=1127.187,5.750,-50.441,179.614,6.431,149.284
C06995=1127.192,5.500,-50.427,179.613,6.427,149.284
C06996=1127.197,5.251,-50.414,179.613,6.422,149.283
C06997=1127.202,5.001,-50.400,179.613,6.418,149.282
C06998=1127.207,4.752,-50.387,179.612,6.413,149.281
C06999=1127.212,4.502,-50.374,179.611,6.409,149.280
C07000=1127.217,4.253,-50.360,179.611,6.404,149.279
C07001=1127.222,4.003,-50.347,179.610,6.399,149.279
C07002=1127.228,3.753,-50.334,179.610,6.395,149.278
C07003=1127.233,3.504,-50.320,179.610,6.391,149.277
C07004=1127.238,3.254,-50.307,179.609,6.386,149.276
C07005=1127.243,3.004,-50.294,179.608,6.382,149.275
C07006=1127.248,2.755,-50.280,179.608,6.378,149.274
C07007=1127.254,2.506,-50.267,179.608,6.373,149.273
C07008=1127.259,2.255,-50.254,179.607,6.368,149.273
C07009=1127.264,2.007,-50.240,179.607,6.364,149.272
C07010=1127.269,1.756,-50.227,179.606,6.359,149.271
C07011=1127.274,1.507,-50.214,179.605,6.355,149.270
C07012=1127.279,1.257,-50.201,179.605,6.351,149.269
C07013=1127.284,1.008,-50.187,179.605,6.346,149.268
C07014=1127.289,0.759,-50.175,179.604,6.341,149.267
C07015=1127.295,0.508,-50.161,179.603,6.337,149.267
C07016=1127.300,0.259,-50.149,179.603,6.332,149.266
C07017=1127.305,0.009,-50.134,179.603,6.328,149.265
C07018=1127.310,-0.240,-50.122,179.602,6.323,149.264
C07019=1127.316,-0.490,-50.109,179.601,6.319,149.264
C07020=1127.320,-0.740,-50.096,179.601,6.314,149.263
C07021=1127.325,-0.989,-50.083,179.600,6.310,149.262
C07022=1127.331,-1.238,-50.069,179.600,6.305,149.261
C07023=1127.335,-1.488,-50.056,179.599,6.301,149.260
C07024=1127.341,-1.738,-50.043,179.599,6.297,149.259
C07025=1127.346,-1.988,-50.030,179.598,6.292,149.258
C07026=1127.351,-2.237,-50.017,179.598,6.287,149.258
C07027=1127.357,-2.487,-50.004,179.597,6.283,149.257
C07028=1127.361,-2.737,-49.991,179.596,6.278,149.256
C07029=1127.367,-2.986,-49.977,179.596,6.273,149.255
C07030=1127.372,-3.235,-49.965,179.595,6.269,149.254
C07031=1127.376,-3.485,-49.952,179.595,6.265,149.254
C07032=1127.382,-3.735,-49.938,179.594,6.260,149.253
C07033=1127.387,-3.984,-49.926,179.594,6.256,149.252
C07034=1127.392,-4.234,-49.913,179.593,6.251,149.251
C07035=1127.398,-4.484,-49.900,179.592,6.247,149.250
C07036=1127.403,-4.733,-49.887,179.592,6.242,149.249
C07037=1127.407,-4.983,-49.874,179.591,6.238,149.249
C07038=1127.413,-5.233,-49.861,179.590,6.233,149.248
C07039=1127.418,-5.482,-49.848,179.590,6.228,149.247
C07040=1127.423,-5.698,-49.837,179.589,6.225,149.246
C07041=1127.427,-5.913,-49.826,179.589,6.221,149.246
C07042=1127.432,-6.128,-49.815,179.588,6.217,149.245
C07043=1127.436,-6.344,-49.803,179.588,6.213,149.244
C07044=1127.440,-6.559,-49.793,179.587,6.209,149.244
C07045=1127.445,-6.774,-49.782,179.587,6.205,149.243
C07046=1127.449,-6.990,-49.771,179.586,6.201,149.242
C07047=1127.454,-7.205,-49.760,179.585,6.197,149.241
C07048=1127.459,-7.455,-49.747,179.585,6.192,149.241
C07049=1127.465,-7.704,-49.734,179.584,6.188,149.240
C07050=1127.469,-7.954,-49.721,179.583,6.183,149.239
C07051=1127.474,-8.204,-49.708,179.583,6.178,149.238
C07052=1127.480,-8.453,-49.696,179.582,6.174,149.238
C07053=1127.485,-8.702,-49.683,179.581,6.169,149.237
C07054=1127.490,-8.953,-49.670,179.581,6.165,149.236
C07055=1127.495,-9.203,-49.658,179.580,6.160,149.235
C07056=1127.500,-9.452,-49.645,179.579,6.156,149.234
C07057=1127.506,-9.701,-49.633,179.578,6.151,149.234
C07058=1127.511,-9.951,-49.620,179.578,6.147,149.233
C07059=1127.516,-10.201,-49.606,179.577,6.142,149.232
C07060=1127.521,-10.450,-49.594,179.576,6.137,149.231
C07061=1127.527,-10.700,-49.582,179.576,6.133,149.230
C07062=1127.532,-10.949,-49.569,179.575,6.128,149.229
C07063=1127.537,-11.199,-49.557,179.574,6.124,149.229
C07064=1127.541,-11.449,-49.544,179.574,6.119,149.228
C07065=1127.546,-11.698,-49.531,179.573,6.114,149.227
C07066=1127.553,-11.948,-49.519,179.572,6.110,149.226
C07067=1127.558,-12.198,-49.506,179.572,6.105,149.225
C07068=1127.563,-12.447,-49.493,179.571,6.100,149.224
C07069=1127.567,-12.697,-49.481,179.570,6.096,149.224
C07070=1127.573,-12.947,-49.469,179.570,6.091,149.223
C07071=1127.578,-13.196,-49.456,179.569,6.087,149.222
C07072=1127.583,-13.446,-49.443,179.568,6.082,149.221
C07073=1127.588,-13.696,-49.432,179.568,6.077,149.220
C07074=1127.594,-13.945,-49.419,179.567,6.073,149.220
C07075=1127.599,-14.194,-49.406,179.566,6.068,149.219
C07076=1127.604,-14.445,-49.394,179.565,6.063,149.218
C07077=1127.609,-14.694,-49.381,179.564,6.059,149.217
C07078=1127.614,-14.943,-49.369,179.564,6.054,149.216
C07079=1127.619,-15.193,-49.357,179.563,6.049,149.216
C07080=1127.624,-15.443,-49.344,179.562,6.045,149.215
C07081=1127.629,-15.692,-49.332,179.562,6.040,149.214
C07082=1127.635,-15.942,-49.320,179.561,6.035,149.213
C07083=1127.640,-16.191,-49.307,179.560,6.030,149.213
C07084=1127.645,-16.441,-49.295,179.559,6.025,149.212
C07085=1127.650,-16.691,-49.282,179.559,6.021,149.211
C07086=1127.655,-16.941,-49.271,179.558,6.016,149.210
C07087=1127.661,-17.190,-49.258,179.557,6.012,149.209
C07088=1127.666,-17.440,-49.246,179.557,6.007,149.208
C07089=1127.671,-17.690,-49.233,179.555,6.002,149.208
C07090=1127.676,-17.939,-49.221,179.555,5.997,149.207
C07091=1127.682,-18.189,-49.209,179.554,5.992,149.206
C07092=1127.687,-18.438,-49.196,179.553,5.988,149.205
C07093=1127.692,-18.688,-49.185,179.553,5.983,149.204
C07094=1127.698,-18.938,-49.173,179.552,5.978,149.203
C07095=1127.703,-19.188,-49.160,179.551,5.973,149.203
C07096=1127.707,-19.403,-49.149,179.550,5.969,149.202
C07097=1127.712,-19.618,-49.139,179.550,5.965,149.201
C07098=1127.716,-19.834,-49.128,179.549,5.961,149.201
C07099=1127.720,-20.049,-49.118,179.548,5.956,149.200
C07100=1127.725,-20.266,-49.108,179.548,5.952,149.199
C07101=1127.730,-20.481,-49.097,179.547,5.948,149.198
C07102=1127.734,-20.696,-49.087,179.546,5.944,149.198
C07103=1127.739,-20.911,-49.076,179.546,5.940,149.197
C07104=1127.744,-21.161,-49.064,179.545,5.935,149.196
C07105=1127.749,-21.410,-49.052,179.544,5.930,149.195
C07106=1127.754,-21.660,-49.040,179.543,5.925,149.195
C07107=1127.760,-21.910,-49.029,179.543,5.921,149.194
C07108=1127.765,-22.160,-49.016,179.542,5.915,149.193
C07109=1127.770,-22.410,-49.004,179.541,5.910,149.192
C07110=1127.776,-22.659,-48.992,179.540,5.906,149.191
C07111=1127.780,-22.908,-48.980,179.539,5.901,149.190
C07112=1127.786,-23.158,-48.968,179.539,5.896,149.189
C07113=1127.791,-23.408,-48.956,179.538,5.891,149.189
C07114=1127.796,-23.658,-48.944,179.537,5.886,149.188
C07115=1127.801,-23.908,-48.932,179.536,5.881,149.187
C07116=1127.806,-24.157,-48.921,179.535,5.876,149.186
C07117=1127.812,-24.407,-48.909,179.534,5.871,149.185
C07118=1127.817,-24.656,-48.896,179.534,5.866,149.184
C07119=1127.823,-24.906,-48.885,179.532,5.861,149.184
C07120=1127.827,-25.155,-48.873,179.532,5.856,149.183
C07121=1127.833,-25.405,-48.861,179.531,5.851,149.182
C07122=1127.838,-25.655,-48.850,179.530,5.846,149.181
C07123=1127.843,-25.904,-48.838,179.530,5.841,149.180
C07124=1127.848,-26.154,-48.826,179.529,5.837,149.179
C07125=1127.854,-26.404,-48.814,179.531,5.833,149.178
C07126=1127.859,-26.654,-48.802,179.532,5.829,149.177
C07127=1127.864,-26.904,-48.791,179.533,5.825,149.176
C07128=1127.869,-27.154,-48.779,179.534,5.821,149.174
C07129=1127.875,-27.402,-48.767,179.535,5.817,149.173
C07130=1127.880,-27.652,-48.755,179.536,5.813,149.172
C07131=1127.885,-27.902,-48.743,179.537,5.809,149.171
C07132=1127.890,-28.152,-48.731,179.537,5.806,149.170
C07133=1127.895,-28.401,-48.720,179.538,5.801,149.169
C07134=1127.901,-28.651,-48.708,179.539,5.798,149.168
C07135=1127.906,-28.901,-48.696,179.540,5.794,149.167
C07136=1127.911,-29.151,-48.685,179.540,5.790,149.166
C07137=1127.916,-29.400,-48.673,179.541,5.785,149.165
C07138=1127.922,-29.649,-48.661,179.541,5.781,149.164
C07139=1127.926,-29.899,-48.650,179.541,5.777,149.163
C07140=1127.932,-30.149,-48.638,179.542,5.773,149.162
C07141=1127.937,-30.399,-48.626,179.542,5.769,149.161
C07142=1127.942,-30.649,-48.615,179.542,5.765,149.160
C07143=1127.947,-30.898,-48.603,179.543,5.761,149.159
C07144=1127.953,-31.148,-48.591,179.543,5.757,149.158
C07145=1127.958,-31.397,-48.580,179.543,5.753,149.157
C07146=1127.964,-31.647,-48.568,179.543,5.748,149.156
C07147=1127.968,-31.897,-48.557,179.543,5.744,149.155
C07148=1127.974,-32.147,-48.545,179.543,5.740,149.154
C07149=1127.979,-32.397,-48.533,179.543,5.735,149.153
C07150=1127.984,-32.646,-48.521,179.543,5.731,149.152
C07151=1127.990,-32.895,-48.509,179.542,5.726,149.151
C07152=1127.994,-33.135,-48.498,179.542,5.723,149.150
C07153=1128.000,-33.374,-48.487,179.542,5.718,149.150
C07154=1128.004,-33.612,-48.476,179.542,5.714,149.149
C07155=1128.009,-33.852,-48.465,179.541,5.709,149.148
C07156=1128.014,-34.092,-48.454,179.541,5.705,149.147
C07157=1128.020,-34.331,-48.443,179.540,5.701,149.146
C07158=1128.025,-34.569,-48.432,179.540,5.696,149.146
C07159=1128.029,-34.809,-48.421,179.539,5.692,149.145
C07160=1128.035,-35.058,-48.410,179.539,5.687,149.144
C07161=1128.040,-35.308,-48.398,179.538,5.683,149.143
C07162=1128.045,-35.558,-48.387,179.537,5.678,149.142
C07163=1128.050,-35.807,-48.375,179.537,5.673,149.141
C07164=1128.056,-36.057,-48.364,179.535,5.668,149.141
C07165=1128.061,-36.307,-48.353,179.535,5.664,149.140
C07166=1128.066,-36.557,-48.341,179.534,5.659,149.139
C07167=1128.071,-36.806,-48.330,179.533,5.654,149.138
C07168=1128.077,-37.056,-48.318,179.532,5.649,149.138
C07169=1128.082,-37.305,-48.307,179.531,5.644,149.137
C07170=1128.087,-37.555,-48.295,179.529,5.639,149.136
C07171=1128.092,-37.805,-48.284,179.528,5.634,149.135
C07172=1128.098,-38.055,-48.273,179.527,5.629,149.135
C07173=1128.103,-38.304,-48.262,179.526,5.624,149.134
C07174=1128.108,-38.554,-48.250,179.524,5.618,149.133
C07175=1128.114,-38.803,-48.239,179.523,5.613,149.133
C07176=1128.119,-39.054,-48.228,179.522,5.608,149.132
C07177=1128.124,-39.303,-48.217,179.520,5.603,149.131
C07178=1128.129,-39.552,-48.206,179.519,5.597,149.130
C07179=1128.135,-39.802,-48.194,179.517,5.592,149.130
C07180=1128.140,-40.053,-48.183,179.516,5.587,149.129
C07181=1128.146,-40.302,-48.172,179.514,5.581,149.128
C07182=1128.151,-40.551,-48.160,179.512,5.576,149.128
C07183=1128.156,-40.802,-48.150,179.511,5.570,149.127
C07184=1128.162,-41.051,-48.138,179.509,5.564,149.126
C07185=1128.166,-41.300,-48.127,179.507,5.559,149.126
C07186=1128.171,-41.551,-48.116,179.505,5.553,149.125
C07187=1128.177,-41.800,-48.105,179.503,5.547,149.124
C07188=1128.182,-42.050,-48.094,179.502,5.542,149.123
C07189=1128.188,-42.299,-48.083,179.500,5.536,149.123
C07190=1128.192,-42.549,-48.072,179.498,5.530,149.122
C07191=1128.198,-42.799,-48.061,179.495,5.524,149.121
C07192=1128.203,-43.048,-48.050,179.493,5.518,149.121
C07193=1128.208,-43.298,-48.040,179.492,5.512,149.120
C07194=1128.214,-43.547,-48.029,179.492,5.508,149.119
C07195=1128.219,-43.798,-48.017,179.492,5.503,149.118
C07196=1128.224,-44.048,-48.006,179.493,5.498,149.117
C07197=1128.230,-44.297,-47.996,179.493,5.494,149.115
C07198=1128.234,-44.547,-47.985,179.493,5.489,149.115
C07199=1128.241,-44.797,-47.974,179.493,5.485,149.113
C07200=1128.245,-45.046,-47.963,179.493,5.480,149.112
C07201=1128.251,-45.296,-47.952,179.494,5.474,149.111
C07202=1128.256,-45.546,-47.942,179.494,5.470,149.110
C07203=1128.261,-45.795,-47.931,179.494,5.465,149.109
C07204=1128.285,-46.882,-47.883,179.075,6.264,149.406
C07205=1128.288,-47.099,-47.874,179.073,6.263,149.407
C07206=1128.294,-47.316,-47.864,179.072,6.263,149.407
C07207=1128.298,-47.534,-47.854,179.069,6.262,149.408
C07208=1128.303,-47.784,-47.843,179.067,6.261,149.408
C07209=1128.308,-48.033,-47.833,179.065,6.260,149.409
C07210=1128.314,-48.283,-47.821,179.063,6.260,149.409
C07211=1128.319,-48.533,-47.811,179.061,6.259,149.409
C07212=1128.324,-48.783,-47.799,179.058,6.259,149.410
C07213=1128.330,-49.032,-47.789,179.056,6.258,149.411
C07214=1128.335,-49.282,-47.777,179.054,6.257,149.411
C07215=1128.340,-49.532,-47.767,179.051,6.256,149.412
C07216=1128.345,-49.781,-47.756,179.049,6.255,149.412
C07217=1128.350,-50.031,-47.745,179.047,6.255,149.413
C07218=1128.356,-50.281,-47.734,179.044,6.254,149.413
C07219=1128.361,-50.531,-47.723,179.042,6.254,149.414
C07220=1128.368,-50.801,-47.711,179.040,6.253,149.414
C07221=1128.373,-51.072,-47.700,179.037,6.252,149.415
C07222=1128.378,-51.344,-47.688,179.035,6.252,149.415
C07223=1128.385,-51.614,-47.676,179.032,6.251,149.416
C07224=1128.390,-51.864,-47.666,179.030,6.251,149.417
C07225=1128.395,-52.113,-47.655,179.028,6.250,149.417
C07226=1128.400,-52.363,-47.644,179.026,6.249,149.418
C07227=1128.405,-52.612,-47.633,179.024,6.248,149.418
C07228=1128.410,-52.862,-47.623,179.021,6.248,149.419
C07229=1128.416,-53.113,-47.611,179.019,6.247,149.419
C07230=1128.421,-53.362,-47.600,179.017,6.247,149.420
C07231=1128.426,-53.612,-47.590,179.015,6.246,149.420
C07232=1128.432,-53.862,-47.580,179.013,6.246,149.421
C07233=1128.437,-54.111,-47.568,179.010,6.245,149.421
C07234=1128.442,-54.361,-47.558,179.008,6.244,149.422
C07235=1128.447,-54.611,-47.548,179.006,6.244,149.422
C07236=1128.452,-54.860,-47.537,179.004,6.243,149.423
C07237=1128.458,-55.111,-47.526,179.001,6.242,149.423
C07238=1128.464,-55.360,-47.515,178.999,6.242,149.424
C07239=1128.469,-55.609,-47.504,178.997,6.241,149.424
C07240=1128.474,-55.859,-47.494,178.994,6.240,149.425
C07241=1128.480,-56.109,-47.484,178.993,6.240,149.425
C07242=1128.484,-56.358,-47.472,178.991,6.239,149.426
C07243=1128.490,-56.608,-47.462,178.988,6.239,149.427
C07244=1128.495,-56.858,-47.452,178.986,6.238,149.427
C07245=1128.501,-57.108,-47.441,178.984,6.238,149.428
C07246=1128.505,-57.357,-47.430,178.981,6.237,149.428
C07247=1128.511,-57.607,-47.420,178.979,6.236,149.429
C07248=1128.516,-57.857,-47.409,178.977,6.236,149.429
C07249=1128.521,-58.107,-47.399,178.974,6.235,149.430
C07250=1128.526,-58.356,-47.388,178.972,6.234,149.430
C07251=1128.532,-58.606,-47.378,178.971,6.234,149.431
C07252=1128.537,-58.855,-47.367,178.968,6.233,149.431
C07253=1128.542,-59.106,-47.357,178.966,6.233,149.432
C07254=1128.548,-59.355,-47.347,178.963,6.232,149.432
C07255=1128.553,-59.605,-47.335,178.961,6.232,149.433
C07256=1128.558,-59.854,-47.325,178.959,6.231,149.433
C07257=1128.563,-60.105,-47.314,178.957,6.230,149.434
C07258=1128.569,-60.354,-47.304,178.955,6.229,149.434
C07259=1128.574,-60.604,-47.294,178.953,6.230,149.435
C07260=1128.579,-60.853,-47.283,178.950,6.229,149.435
C07261=1128.585,-61.103,-47.273,178.948,6.228,149.436
C07262=1128.590,-61.353,-47.262,178.946,6.227,149.436
C07263=1128.595,-61.603,-47.252,178.944,6.227,149.437
C07264=1128.601,-61.852,-47.242,178.942,6.226,149.437
C07265=1128.606,-62.102,-47.231,178.939,6.225,149.438
C07266=1128.611,-62.352,-47.221,178.937,6.225,149.439
C07267=1128.616,-62.602,-47.210,178.935,6.225,149.439
C07268=1128.622,-62.852,-47.200,178.933,6.224,149.440
C07269=1128.627,-63.101,-47.189,178.931,6.223,149.440
C07270=1128.632,-63.351,-47.179,178.928,6.223,149.441
C07271=1128.637,-63.600,-47.169,178.926,6.222,149.441
C07272=1128.643,-63.850,-47.159,178.924,6.221,149.442
C07273=1128.648,-64.100,-47.148,178.922,6.221,149.442
C07274=1128.653,-64.350,-47.138,178.920,6.221,149.443
C07275=1128.659,-64.599,-47.128,178.918,6.220,149.443
C07276=1128.664,-64.849,-47.117,178.915,6.219,149.444
C07277=1128.670,-65.099,-47.107,178.913,6.219,149.444
C07278=1128.675,-65.348,-47.097,178.911,6.218,149.445
C07279=1128.680,-65.599,-47.086,178.909,6.217,149.445
C07280=1128.685,-65.848,-47.077,178.906,6.216,149.446
